// TwinCAT 3 PLC project PLC
// ProgramVersion: 3.1.4023.0
// libraries:
//   Tc2_MC2, * (Beckhoff Automation GmbH)
//   Tc2_MC2_Drive, * (Beckhoff Automation GmbH)
//   Tc2_Standard, * (Beckhoff Automation GmbH)
//   Tc2_System, * (Beckhoff Automation GmbH)
//   Tc2_TcpIp, * (Beckhoff Automation GmbH)
//   Tc2_Utilities, * (Beckhoff Automation GmbH)
//   Tc3_Database, * (Beckhoff Automation GmbH)
//   Tc3_EventLogger, * (Beckhoff Automation GmbH)
//   Tc3_Module, * (Beckhoff Automation GmbH)
// project tree:
//   DUTs/ConveyorSystem/ ST_CPI_Module.TcDUT
//   DUTs/OPC_UA/ OPC_CNC_Data_Collection.TcDUT
//   DUTs/PyADS/ ST_PyADS_Test.TcDUT
//   DUTs/RGB/ ST_RGB_In.TcDUT, ST_RGB_Light.TcDUT, ST_RGB_Out.TcDUT
//   DUTs/ ST_Dut_Data.TcDUT
//   DUTs/Vise/ E_ViseSocketState.TcDUT, E_Vise_State.TcDUT, E_Vise_Command.TcDUT, ST_Order.TcDUT, ST_Vise_Sensors.TcDUT, ST_Vise_Status.TcDUT
//   DUTs/Executer/ E_Executer_State.TcDUT
//   GVLs/ GVL_Ads.TcGVL, GVL_CNC1.TcGVL, GVL_CNC2.TcGVL, GVL_CNC3.TcGVL, GVL_Constant.TcGVL, GVL_ConveyorSystem.TcGVL, GVL_IO.TcGVL, GVL_IO_CNC1.TcGVL, GVL_Main.TcGVL, GVL_Palette.TcGVL, GVL_Python.TcGVL, GVL_RFID.TcGVL, GVL_Safety.TcGVL
//   / PlcTask.TcTTO
//   POUs/ Blink.TcPOU, ConveyorSystem.TcPOU, InitTCPIP.TcPOU, MAIN.TcPOU, SafetyPRG.TcPOU, SQL_Test.TcPOU, Test.TcPOU
//   POUs/CNC_1/ CNC_1.TcPOU
//   POUs/CNC_2/ CNC_2.TcPOU
//   POUs/CNC_3/ CNC_3.TcPOU
//   POUs/FBs/AWEA/DUTs/ ST_AWEA_In.TcDUT, ST_AWEA_Out.TcDUT
//   POUs/FBs/AWEA/ FB_AWEA.TcPOU
//   POUs/FBs/BTL/DUTs/ U_to_dint.TcDUT
//   POUs/FBs/BTL/ FB_BTL1AR0.TcPOU
//   POUs/FBs/Camera/ FB_TCP_IP_Comm.TcPOU
//   POUs/FBs/CNC_Servo/DUTs/ E_CncServoCommand.TcTLEO
//   POUs/FBs/CNC_Servo/ FB_CNC_Servo.TcPOU
//   POUs/FBs/FanucCNC/DUTs/ E_CNC_Robot_Command.TcDUT, E_CNC_Robot_Path.TcTLEO, E_CNC_Robot_Programs.TcTLEO, E_Lifter.TcDUT, ST_CNC_Robot_Control.TcDUT, ST_CNC_Robot_Status.TcDUT, U_CNC_Fanuc_Input.TcDUT, U_CNC_Fanuc_Output.TcDUT
//   POUs/FBs/FanucCNC/ FB_Fanuc_CNC.TcPOU
//   POUs/FBs/FanucKardex/DUTs/ E_Kardex_Robot_Command.TcDUT, E_Kardex_Robot_Programs.TcTLEO, ST_Kardex_Robot_Control.TcDUT, ST_Kardex_Robot_Status.TcDUT, U_Kardex_Fanuc_Input.TcDUT, U_Kardex_Fanuc_Output.TcDUT
//   POUs/FBs/FanucKardex/ FB_Fanuc_Kardex.TcPOU
//   POUs/FBs/Fanuc/DUTs/ E_Robot_Command.TcDUT, E_Robot_Programs.TcTLEO, ST_Robot_Control.TcDUT (not stored), ST_Robot_Status.TcDUT, U_Fanuc_Input.TcDUT, U_Fanuc_Output.TcDUT
//   POUs/FBs/Fanuc/ FB_Fanuc.TcPOU
//   POUs/FBs/ FB_Conveyor.TcPOU, FB_Door.TcPOU, FB_Server.TcPOU, FB_SQL.TcPOU, FB_Vise_Station.TcPOU
//   POUs/FBs/ID200/DUTs/ E_CarrierType.TcTLEO, E_Command.TcTLEO, E_TagStatus.TcTLEO, RawToUlint.TcDUT, ST_Active_RFIDs.TcDUT, ST_Tag_Data.TcDUT, WordToBytes.TcDUT
//   POUs/FBs/ID200/ FB_ID200.TcPOU
//   POUs/FBs/Lift/ FB_Lift.TcPOU
//   POUs/FBs/MPS/DUTs/ U_to_int.TcDUT
//   POUs/FBs/MPS/ FB_MPS100.TcPOU
//   POUs/FBs/MySQL/NextVise/DUTs/ ST_ParaVal_GetNextVise.TcDUT
//   POUs/FBs/MySQL/NextVise/ FB_SP_spGetNextVise.TcPOU
//   POUs/FBs/MySQL/SetViseState/DUTs/ ST_ParaVal_SetViseStae.TcDUT
//   POUs/FBs/MySQL/SetViseState/ FB_SP_spSetViseStae.TcPOU
//   POUs/FBs/MySQL/UpdateVise/DUTs/ ST_ParaVal_UpdateVise.TcDUT
//   POUs/FBs/MySQL/UpdateVise/ FB_SP_spUpdateVise.TcPOU
//   POUs/FBs/Pneumatics/ FB_Bistabil.TcPOU, FB_Stopper.TcPOU, FB_Stopper2.TcPOU
//   POUs/FBs/Router/ FB_Router.TcPOU
//   POUs/FBs/ServoVise/DUTs/ E_ServoVise_Command.TcTLEO, E_ViseJawState.TcTLEO
//   POUs/FBs/ServoVise/ FB_ServoVise.TcPOU, FB_TorqueCheck.TcPOU
//   POUs/FBs/Utilities/ FB_CommandLineExecuter.TcPOU, FB_FullCycleTime.TcPOU, FB_GenPulse.TcPOU, FB_Not_SmartLight.TcPOU, FB_RGB_Light.TcPOU, FB_TcEvent.TcPOU, FB_UpsC69xx.TcPOU, FB_UserLed.TcPOU, FB_WorkLight.TcPOU
//   POUs/Robot7AxisStation/ Robot7AxisProgram.TcPOU
//   POUs/RobotKardexStation/ RobotKardexProgram.TcPOU
//   POUs/RobotViseStation/ RobotCncProgram.TcPOU, ViseProgram.TcPOU
//   POUs/Temp/Fanuc/ E_Fanuc_Program.TcDUT, ST_FanucReq.TcDUT, ST_Fanuc_Alarm_In.TcDUT, ST_Fanuc_Alarm_Out.TcDUT, ST_Fanuc_Area_In.TcDUT, ST_Fanuc_Control_In.TcDUT, ST_Fanuc_Control_Out.TcDUT, ST_Fanuc_Data_In.TcDUT, ST_Fanuc_Data_Out.TcDUT, ST_Fanuc_DIO_In.TcDUT, ST_Fanuc_Emergency_In.TcDUT, ST_Fanuc_HandShake_In.TcDUT, ST_Fanuc_Handshake_Out.TcDUT, ST_Fanuc_In.TcDUT, ST_Fanuc_ManPos.TcDUT, ST_Fanuc_Out.TcDUT, ST_Fanuc_Press_Out.TcDUT, ST_Fanuc_Prog_In.TcDUT, ST_Fanuc_Prog_Out.TcDUT, U_Fanuc_In.TcDUT, U_Fanuc_Out.TcDUT
//   POUs/Temp/ FB_ContiRobot.TcPOU, Robot.TcPOU
//   POUs/UploadingStation/ UploadingProgram.TcPOU
// real-time tasks:
//   TASK PlcTask: cycle T#10ms, priority 20, ADS port 350
//   TASK ProfiNET: cycle T#16ms, priority 25, ADS port 351
//   TASK Job Task: cycle default, priority 32
// motion (NC):
//   TASK NC-Task 1 SAF: cycle T#2ms, priority 4, ADS port 501
//   TASK NC-Task 1 SVB: cycle T#10ms, priority 8, ADS port 511
//   AXIS Axis 1 (id 1)
//     Dynamic: Acceleration=6.6163, Deceleration=6.6163, Jerk=19.8489
//     Velo: RefSearch=0.044108688151042, RefSync=0.044108688151042, SlowManual=0.220543440755208, FastManual=4, Fast=4.41086881510417, Maximum=4.41087
//     OtherSettings: AllowMotionCmdToSlave=true
//     encoder EncType=8
//       EncPara: ScaleFactorNumerator=0.04, ScaleFactorDenominator=1048576, MaxCount=#xffffffff
//         TimeComp: TimeCompMode=1
//     drive DrvType=9
//       DrvPara: MaxCount=#xffffffff, DriveControlDWord=#x00030100
//         Analog: VeloReferenz=4.85195569661458, VeloScale=1.02400649589962, TorqueSetpointScale=10, ScaleFactorActTorque=0.1
//         TimeComp: TaskDelayCycles=1
//     controller CtrType=1
//       CtrPara: PriorControlFactor=1
//         Observer: BandWidth=20
//   AXIS Axis 2 (id 2)
//     Dynamic: Acceleration=6.6163, Deceleration=6.6163, Jerk=19.8489
//     Velo: RefSearch=0.044108688151042, RefSync=0.044108688151042, SlowManual=0.220543440755208, FastManual=4, Fast=4.41086881510417, Maximum=4.41087
//     OtherSettings: AllowMotionCmdToSlave=true
//     encoder EncType=8
//       EncPara: ScaleFactorNumerator=0.04, ScaleFactorDenominator=1048576, MaxCount=#xffffffff
//         TimeComp: TimeCompMode=1
//     drive DrvType=9
//       DrvPara: MaxCount=#xffffffff, DriveControlDWord=#x00030100
//         Analog: VeloReferenz=4.85195569661458, VeloScale=1.02400649589962, TorqueSetpointScale=10, ScaleFactorActTorque=0.1
//         TimeComp: TaskDelayCycles=1
//     controller CtrType=1
//       CtrPara: PriorControlFactor=1
//         Observer: BandWidth=20
//   AXIS Axis 3 (id 3)
//     Dynamic: Acceleration=6.6163, Deceleration=6.6163, Jerk=19.8489
//     Velo: RefSearch=0.044108688151042, RefSync=0.044108688151042, SlowManual=0.220543440755208, FastManual=4, Fast=4.41086881510417, Maximum=4.41087
//     OtherSettings: AllowMotionCmdToSlave=true
//     encoder EncType=8
//       EncPara: ScaleFactorNumerator=0.04, ScaleFactorDenominator=1048576, MaxCount=#xffffffff
//         TimeComp: TimeCompMode=1
//     drive DrvType=9
//       DrvPara: MaxCount=#xffffffff, DriveControlDWord=#x00030100
//         Analog: VeloReferenz=4.85195569661458, VeloScale=1.02400649589962, TorqueSetpointScale=10, ScaleFactorActTorque=0.1
//         TimeComp: TaskDelayCycles=1
//     controller CtrType=1
//       CtrPara: PriorControlFactor=1
//         Observer: BandWidth=20
// I/O:
//   DEVICE Device 1 (RT-Ethernet Adapter)
//   DEVICE Fanuc_Vise, AmsNetId 192.168.81.10.5.1
//     Box 1 (CU2508) [CU2508 Ethernet Port]
//     Box 2 (FANUC R-30iB V8.20) [FANUC R-30iB V8.20]
//   DEVICE Fanuc_7Axis, AmsNetId 192.168.81.10.6.1
//     Box 3 (CU2508) [CU2508 Ethernet Port]
//     Box 4 (FANUC R-30iB V8.20) [FANUC R-30iB V8.20]
//   DEVICE Fanuc_Kardex, AmsNetId 192.168.81.10.7.1
//     Box 5 (CU2508) [CU2508 Ethernet Port]
//     Box 6 (FANUC R-30iB V8.20) [FANUC R-30iB V8.20]
//   DEVICE CNC_1, AmsNetId 192.168.81.10.8.1
//     Box 7 (CU2508) [CU2508 Ethernet Port]
//     Drive 9 (AX5106-0000-0214) [AX5106-0000-0214 EtherCAT Drive (SoE, 1 Ch.)]
//       Term 16 (AX5805) [AX5805 (Safety Drive Option)]
//         modules: Module 1 (Safety Process Data, 1 axis), Module 2 (Standard Process Data, 1 axis)
//       Term 18 (EL9011) [EL9011 End Terminal]
//     Box 10 (BNI ECT-508-105-Z015) [BNI ECT-508-105-Z015 (BNI0077)]
//       modules: Module 1 (IOL_I_4byte), Module 2 (STD_IN_1bit), Module 3 (STD_IN_1bit), Module 4 (STD_IN_1bit), Module 5 (STD_IN_1bit), Module 6 (STD_IN_1bit), Module 7 (STD_IN_1bit), Module 8 (STD_IN_1bit)
//     Term 11 (EK1100) [EK1100 EtherCAT Coupler (2A E-Bus)]
//       Term 12 (EL6910) [EL6910, TwinSAFE PLC]
//       Term 13 (EL1809) [EL1809 16Ch. Dig. Input 24V, 3ms]
//       Term 14 (EL2809-0015) [EL2809-0015 16Ch. Dig. Output 24V DC, 0.35A, not short-circuit proof]
//       Term 11 (EL9011) [EL9011 End Terminal]
//     Box 15 (EP1957-0022) [EP1957, 8Ch. Safety Input 24V, 4Ch. Safety Output 24V, 0.5A, TwinSAFE]
//       modules: Module 1 (FSOE), Module 2 (FSOUT), Module 3 (DEVICEIO), Module 4 (FSLOGIC)
//   DEVICE CNC_2, AmsNetId 192.168.81.10.9.1
//     Box 18 (CU2508) [CU2508 Ethernet Port]
//     Drive 19 (AX5106-0000-0214) [AX5106-0000-0214 EtherCAT Drive (SoE, 1 Ch.)]
//       Term 20 (AX5805) [AX5805 (Safety Drive Option)]
//         modules: Module 1 (Safety Process Data, 1 axis), Module 2 (Standard Process Data, 1 axis)
//       Term 10 (EL9011) [EL9011 End Terminal]
//     Box 21 (BNI ECT-508-105-Z015) [BNI ECT-508-105-Z015 (BNI0077)]
//       modules: Module 1 (IOL_I_4byte), Module 2 (STD_IN_1bit), Module 3 (STD_IN_1bit), Module 4 (STD_IN_1bit), Module 5 (STD_IN_1bit), Module 6 (STD_IN_1bit), Module 7 (STD_IN_1bit), Module 8 (STD_IN_1bit)
//     Term 22 (EK1100) [EK1100 EtherCAT Coupler (2A E-Bus)]
//       Term 23 (EL6910) [EL6910, TwinSAFE PLC]
//       Term 24 (EL1809) [EL1809 16Ch. Dig. Input 24V, 3ms]
//       Term 25 (EL2809) [EL2809 16Ch. Dig. Output 24V, 0.5A]
//       Term 11 (EL9011) [EL9011 End Terminal]
//     Box 26 (EP1957-0022) [EP1957, 8Ch. Safety Input 24V, 4Ch. Safety Output 24V, 0.5A, TwinSAFE]
//       modules: Module 1 (FSOE), Module 2 (FSOUT), Module 3 (DEVICEIO), Module 4 (FSLOGIC)
//   DEVICE CNC_3, AmsNetId 192.168.81.10.10.1
//     Box 29 (CU2508) [CU2508 Ethernet Port]
//     Drive 30 (AX5106-0000-0214) [AX5106-0000-0214 EtherCAT Drive (SoE, 1 Ch.)]
//       Term 31 (AX5805) [AX5805 (Safety Drive Option)]
//         modules: Module 1 (Safety Process Data, 1 axis), Module 2 (Standard Process Data, 1 axis)
//       Term 10 (EL9011) [EL9011 End Terminal]
//     Box 32 (BNI ECT-508-105-Z015) [BNI ECT-508-105-Z015 (BNI0077)]
//       modules: Module 1 (IOL_I_4byte), Module 2 (STD_IN_1bit), Module 3 (STD_IN_1bit), Module 4 (STD_IN_1bit), Module 5 (STD_IN_1bit), Module 6 (STD_IN_1bit), Module 7 (STD_IN_1bit), Module 8 (STD_IN_1bit)
//     Term 33 (EK1100) [EK1100 EtherCAT Coupler (2A E-Bus)]
//       Term 34 (EL6910) [EL6910, TwinSAFE PLC]
//       Term 35 (EL1809) [EL1809 16Ch. Dig. Input 24V, 3ms]
//       Term 36 (EL2809) [EL2809 16Ch. Dig. Output 24V, 0.5A]
//       Term 11 (EL9011) [EL9011 End Terminal]
//     Box 37 (EP1957-0022) [EP1957, 8Ch. Safety Input 24V, 4Ch. Safety Output 24V, 0.5A, TwinSAFE]
//       modules: Module 1 (FSOE), Module 2 (FSOUT), Module 3 (DEVICEIO), Module 4 (FSLOGIC)
//   DEVICE Main, AmsNetId 192.168.81.10.11.1
//     Box 40 (CU2508) [CU2508 Ethernet Port]
//     Term 41 (EK1100) [EK1100 EtherCAT Coupler (2A E-Bus)]
//       Term 42 (EL6910) [EL6910, TwinSAFE PLC]
//       Term 43 (EL1918) [EL1918, 8Ch. Safety Input 24V, TwinSAFE]
//         modules: Module 1 (FSOE), Module 2 (FSLOGIC)
//       Term 44 (EL1904) [EL1904, 4 Ch. Safety Input 24V, TwinSAFE]
//         modules: Module 1 (FSOES)
//       Term 45 (EL1904) [EL1904, 4 Ch. Safety Input 24V, TwinSAFE]
//         modules: Module 1 (FSOES)
//       Term 46 (EL2904) [EL2904, 4 Ch. Safety Output 24V, 0.5A, TwinSAFE]
//         modules: Module 1 (FSOES), Module 2 (DO)
//       Term 47 (EL2904) [EL2904, 4 Ch. Safety Output 24V, 0.5A, TwinSAFE]
//         modules: Module 1 (FSOES), Module 2 (DO)
//       Term 48 (EL1809) [EL1809 16Ch. Dig. Input 24V, 3ms]
//       Term 49 (EL1809) [EL1809 16Ch. Dig. Input 24V, 3ms]
//       Term 50 (EL1809) [EL1809 16Ch. Dig. Input 24V, 3ms]
//       Term 51 (EL2809) [EL2809 16Ch. Dig. Output 24V, 0.5A]
//       Term 52 (EL2809-0015) [EL2809-0015 16Ch. Dig. Output 24V DC, 0.35A, not short-circuit proof]
//       Term 53 (EL9410) [EL9410 E-Bus Power Supplier  (Diagnostics)]
//       Term 54 (EL2809-0015) [EL2809-0015 16Ch. Dig. Output 24V DC, 0.35A, not short-circuit proof]
//       Term 55 (EL6224) [EL6224 (IO Link Master)]
//       Term 56 (EL6224) [EL6224 (IO Link Master)]
//       Term 18 (EL6631) [EL6631 PROFINET IO Controller]
//       Term 36 (EL9011) [EL9011 End Terminal]
//     Term 58 (EK1100) [EK1100 EtherCAT Coupler (2A E-Bus)]
//       Term 59 (EL1918) [EL1918, 8Ch. Safety Input 24V, TwinSAFE]
//         modules: Module 1 (FSOE), Module 2 (FSLOGIC)
//       Term 60 (EL1918) [EL1918, 8Ch. Safety Input 24V, TwinSAFE]
//         modules: Module 1 (FSOE), Module 2 (FSLOGIC)
//       Term 61 (EL1904) [EL1904, 4 Ch. Safety Input 24V, TwinSAFE]
//         modules: Module 1 (FSOES)
//       Term 62 (EL1904) [EL1904, 4 Ch. Safety Input 24V, TwinSAFE]
//         modules: Module 1 (FSOES)
//       Term 63 (EL2904) [EL2904, 4 Ch. Safety Output 24V, 0.5A, TwinSAFE]
//         modules: Module 1 (FSOES), Module 2 (DO)
//       Term 64 (EL2904) [EL2904, 4 Ch. Safety Output 24V, 0.5A, TwinSAFE]
//         modules: Module 1 (FSOES), Module 2 (DO)
//       Term 65 (EL1809) [EL1809 16Ch. Dig. Input 24V, 3ms]
//       Term 66 (EL1809) [EL1809 16Ch. Dig. Input 24V, 3ms]
//       Term 67 (EL1809) [EL1809 16Ch. Dig. Input 24V, 3ms]
//       Term 68 (EL2809-0015) [EL2809-0015 16Ch. Dig. Output 24V DC, 0.35A, not short-circuit proof]
//       Term 69 (EL2809-0015) [EL2809-0015 16Ch. Dig. Output 24V DC, 0.35A, not short-circuit proof]
//       Term 70 (EL9410) [EL9410 E-Bus Power Supplier  (Diagnostics)]
//       Term 71 (EL2809-0015) [EL2809-0015 16Ch. Dig. Output 24V DC, 0.35A, not short-circuit proof]
//       Term 72 (EL2809-0015) [EL2809-0015 16Ch. Dig. Output 24V DC, 0.35A, not short-circuit proof]
//       Term 34 (EL6614) [EL6614 4 Port Switch (Ethernet, CoE)]
//       Term 37 (EL9011) [EL9011 End Terminal]
//     Box 74 (CPX-FB37) [CPX-FB37 Fieldbus module]
//       modules: Module 1 (FB37-RIO), Module 2 (CPI: 16 Byte I/0 Byte O), Module 3 (CPI: 4 Byte I/0 Byte O), Module 4 (MPA1G VMPA1-FB-EMG-8 [8DO]), Module 5 (MPA1G VMPA1-FB-EMG-8 [8DO]), Module 6 (MPA1G VMPA1-FB-EMG-8 [8DO]), Module 7 (MPA1G VMPA1-FB-EMG-8 [8DO]), Module 8 (MPA1G VMPA1-FB-EMG-8 [8DO]), Module 9 (MPA1G VMPA1-FB-EMG-8 [8DO]), Module 10 (MPA1G VMPA1-FB-EMG-8 [8DO]), Module 11 (MPA1G VMPA1-FB-EMG-8 [8DO]), Module 12 (MPA1G VMPA1-FB-EMG-8 [8DO]), Module 13 (MPA1G VMPA1-FB-EMG-8 [8DO]), Module 14 (MPA1G VMPA1-FB-EMG-8 [8DO])
//     Box 75 (BNI ECT-508-105-Z015) [BNI ECT-508-105-Z015 (BNI0077)]
//       modules: Module 1 (IOL_I_2byte), Module 2 (IOL_I_2byte), Module 3 (STD_IN_1bit), Module 4 (STD_IN_1bit), Module 5 (STD_IN_1bit), Module 6 (STD_IN_1bit), Module 7 (STD_IN_1bit), Module 8 (STD_IN_1bit)
//   DEVICE Vise, AmsNetId 192.168.81.10.12.1
//     Term 77 (EK1100) [EK1100 EtherCAT Coupler (2A E-Bus)]
//       Term 78 (EL6070-0033) [EL6070-0033 1Ch. Licence key terminal, individual licences]
//       Term 79 (EL1918) [EL1918, 8Ch. Safety Input 24V, TwinSAFE]
//         modules: Module 2 (FSLOGIC)
//       Term 109 (EL1904) [EL1904, 4 Ch. Safety Input 24V, TwinSAFE]
//         modules: Module 1 (FSOES)
//       Term 110 (EL1904) [EL1904, 4 Ch. Safety Input 24V, TwinSAFE]
//         modules: Module 1 (FSOES)
//       Term 80 (EL2904) [EL2904, 4 Ch. Safety Output 24V, 0.5A, TwinSAFE]
//         modules: Module 1 (FSOES), Module 2 (DO)
//       Term 81 (EL2904) [EL2904, 4 Ch. Safety Output 24V, 0.5A, TwinSAFE]
//         modules: Module 1 (FSOES), Module 2 (DO)
//       Term 82 (EL1809) [EL1809 16Ch. Dig. Input 24V, 3ms]
//       Term 83 (EL1809) [EL1809 16Ch. Dig. Input 24V, 3ms]
//       Term 84 (EL2809) [EL2809 16Ch. Dig. Output 24V, 0.5A]
//       Term 85 (EL6224) [EL6224 (IO Link Master)]
//       Term 86 (EK1110) [EK1110 EtherCAT extension]
//     Box 87 (EasyCAT_RGB_2x8) [EasyCAT_RGB_2x8]
//     Box 88 (CPX-FB37) [CPX-FB37 Fieldbus module]
//       modules: Module 1 (FB37-RIO), Input, Output1, Output2, Output3, Output4, Output5, Output6, Output7
//     Box 89 (CPX-FB37) [CPX-FB37 Fieldbus module]
//       modules: Module 1 (FB37-RIO), Input, Output1, Output2, Output3, Output4, Output5, Output6, Output7
//     Term 90 (EK1100) [EK1100 EtherCAT Coupler (2A E-Bus)]
//       Term 91 (EL1809) [EL1809 16Ch. Dig. Input 24V, 3ms]
//       Term 92 (EL2809-0015) [EL2809-0015 16Ch. Dig. Output 24V DC, 0.35A, not short-circuit proof]
//       Term 19 (EL9011) [EL9011 End Terminal]
//     Box 93 (EP1957-0022) [EP1957, 8Ch. Safety Input 24V, 4Ch. Safety Output 24V, 0.5A, TwinSAFE]
//       modules: Module 1 (FSOE), Module 2 (FSOUT), Module 3 (DEVICEIO), Module 4 (FSLOGIC)
//     Box 94 (EP1957-0022) [EP1957, 8Ch. Safety Input 24V, 4Ch. Safety Output 24V, 0.5A, TwinSAFE]
//       modules: Module 1 (FSOE), Module 2 (FSOUT), Module 3 (DEVICEIO), Module 4 (FSLOGIC)
//   DEVICE Device 2 (EL6631), AmsNetId 192.168.81.10.3.1
//     rfm1 [Bosch Rexroth DAP1,ID 200/C-ETH, no PDEV 3842410060]
//       modules: Term 1 (DAP Module), Data
//     rfm2 [Bosch Rexroth DAP1,ID 200/C-ETH, no PDEV 3842410060]
//       modules: Term 3 (DAP Module), Data
//     rfm3 [Bosch Rexroth DAP1,ID 200/C-ETH, no PDEV 3842410060]
//       modules: Term 5 (DAP Module), Data
//     rfm4 [Bosch Rexroth DAP1,ID 200/C-ETH, no PDEV 3842410060]
//       modules: Term 7 (DAP Module), Data
//     rfm5 [Bosch Rexroth DAP1,ID 200/C-ETH, no PDEV 3842410060]
//       modules: Term 9 (DAP Module), Data
//     rfm6 [Bosch Rexroth DAP1,ID 200/C-ETH, no PDEV 3842410060]
//       modules: Term 11 (DAP Module), Data
//     rfm7 [Bosch Rexroth DAP1,ID 200/C-ETH, no PDEV 3842410060]
//       modules: Term 13 (DAP Module), Data
//     rfm8 [Bosch Rexroth DAP1,ID 200/C-ETH, no PDEV 3842410060]
//       modules: Term 15 (DAP Module), Data
//     rfm9 [Bosch Rexroth DAP1,ID 200/C-ETH, no PDEV 3842410060]
//       modules: Term 17 (DAP Module), Data
//     rfm10 [Bosch Rexroth DAP1,ID 200/C-ETH, no PDEV 3842410060]
//       modules: Term 19 (DAP Module), Data
// variable links:
//   CNC_1 <-> CNC_1/Drive 9 (AX5106-0000-0214)/Term 16 (AX5805)
//     Term 11 (EK1100)/Term 12 (EL6910)/ConnectionOutputs/Message_3 RxPDO <-> Module 1 (Safety Process Data, 1 axis)/Inputs (Statusword)/FSOE
//   CNC_1 <-> CNC_1/Term 11 (EK1100)/Term 12 (EL6910)
//     Box 15 (EP1957-0022)/Module 1 (FSOE)/FSoE Inputs/FSOE <-> ConnectionOutputs/Message_4 RxPDO
//     Box 15 (EP1957-0022)/Module 1 (FSOE)/FSoE Outputs/FSOE <-> ConnectionInputs/Message_4 TxPDO
//     Drive 9 (AX5106-0000-0214)/Term 16 (AX5805)/Module 1 (Safety Process Data, 1 axis)/Outputs (Controlword)/FSOE <-> ConnectionInputs/Message_3 TxPDO
//   CNC_1 <-> Main/Term 41 (EK1100)/Term 42 (EL6910)
//     Term 11 (EK1100)/Term 12 (EL6910)/ConnectionInputs/Message_18 TxPDO <-> ConnectionOutputs/Message_26 RxPDO
//     Term 11 (EK1100)/Term 12 (EL6910)/ConnectionOutputs/Message_18 RxPDO <-> ConnectionInputs/Message_26 TxPDO
//   CNC_2 <-> CNC_2/Box 26 (EP1957-0022)
//     Term 22 (EK1100)/Term 23 (EL6910)/ConnectionOutputs/Message_8 RxPDO <-> Module 1 (FSOE)/FSoE Inputs/FSOE
//   CNC_2 <-> CNC_2/Drive 19 (AX5106-0000-0214)/Term 20 (AX5805)
//     Term 22 (EK1100)/Term 23 (EL6910)/ConnectionInputs/Message_7 TxPDO <-> Module 1 (Safety Process Data, 1 axis)/Outputs (Controlword)/FSOE
//     Term 22 (EK1100)/Term 23 (EL6910)/ConnectionOutputs/Message_7 RxPDO <-> Module 1 (Safety Process Data, 1 axis)/Inputs (Statusword)/FSOE
//   CNC_2 <-> CNC_2/Term 22 (EK1100)/Term 23 (EL6910)
//     Box 26 (EP1957-0022)/Module 1 (FSOE)/FSoE Outputs/FSOE <-> ConnectionInputs/Message_8 TxPDO
//   CNC_2 <-> Main/Term 41 (EK1100)/Term 42 (EL6910)
//     Term 22 (EK1100)/Term 23 (EL6910)/ConnectionOutputs/Message_9 RxPDO <-> ConnectionInputs/Message_28 TxPDO
//   CNC_3 <-> CNC_3/Box 37 (EP1957-0022)
//     Term 33 (EK1100)/Term 34 (EL6910)/ConnectionOutputs/Message_9 RxPDO <-> Module 1 (FSOE)/FSoE Inputs/FSOE
//   CNC_3 <-> CNC_3/Drive 30 (AX5106-0000-0214)/Term 31 (AX5805)
//     Term 33 (EK1100)/Term 34 (EL6910)/ConnectionInputs/Message_8 TxPDO <-> Module 1 (Safety Process Data, 1 axis)/Outputs (Controlword)/FSOE
//     Term 33 (EK1100)/Term 34 (EL6910)/ConnectionOutputs/Message_8 RxPDO <-> Module 1 (Safety Process Data, 1 axis)/Inputs (Statusword)/FSOE
//   CNC_3 <-> CNC_3/Term 33 (EK1100)/Term 34 (EL6910)
//     Box 37 (EP1957-0022)/Module 1 (FSOE)/FSoE Outputs/FSOE <-> ConnectionInputs/Message_9 TxPDO
//   CNC_3 <-> Main/Term 41 (EK1100)/Term 42 (EL6910)
//     Term 33 (EK1100)/Term 34 (EL6910)/ConnectionOutputs/Message_10 RxPDO <-> ConnectionInputs/Message_29 TxPDO
//   Main <-> CNC_2/Term 22 (EK1100)/Term 23 (EL6910)
//     Term 41 (EK1100)/Term 42 (EL6910)/ConnectionOutputs/Message_28 RxPDO <-> ConnectionInputs/Message_9 TxPDO
//   Main <-> CNC_3/Term 33 (EK1100)/Term 34 (EL6910)
//     Term 41 (EK1100)/Term 42 (EL6910)/ConnectionOutputs/Message_29 RxPDO <-> ConnectionInputs/Message_10 TxPDO
//   Main <-> Main/Term 41 (EK1100)/Term 42 (EL6910)
//     Term 41 (EK1100)/Term 43 (EL1918)/Module 1 (FSOE)/FSoE Outputs/FSOE <-> ConnectionInputs/Message_17 TxPDO
//     Term 41 (EK1100)/Term 44 (EL1904)/Module 1 (FSOES)/RxPDO/FSOE <-> ConnectionInputs/Message_3 TxPDO
//     Term 41 (EK1100)/Term 45 (EL1904)/Module 1 (FSOES)/RxPDO/FSOE <-> ConnectionInputs/Message_18 TxPDO
//     Term 41 (EK1100)/Term 46 (EL2904)/Module 1 (FSOES)/RxPDO/FSOE <-> ConnectionInputs/Message_5 TxPDO
//     Term 41 (EK1100)/Term 44 (EL1904)/Module 1 (FSOES)/TxPDO/FSOE <-> ConnectionOutputs/Message_3 RxPDO
//     Term 41 (EK1100)/Term 45 (EL1904)/Module 1 (FSOES)/TxPDO/FSOE <-> ConnectionOutputs/Message_18 RxPDO
//     Term 41 (EK1100)/Term 47 (EL2904)/Module 1 (FSOES)/TxPDO/FSOE <-> ConnectionOutputs/Message_22 RxPDO
//   Main <-> Main/Term 41 (EK1100)/Term 43 (EL1918)
//     Term 41 (EK1100)/Term 42 (EL6910)/ConnectionOutputs/Message_17 RxPDO <-> Module 1 (FSOE)/FSoE Inputs/FSOE
//   Main <-> Main/Term 41 (EK1100)/Term 46 (EL2904)
//     Term 41 (EK1100)/Term 42 (EL6910)/ConnectionOutputs/Message_5 RxPDO <-> Module 1 (FSOES)/TxPDO/FSOE
//   Main <-> Main/Term 41 (EK1100)/Term 47 (EL2904)
//     Term 41 (EK1100)/Term 42 (EL6910)/ConnectionInputs/Message_22 TxPDO <-> Module 1 (FSOES)/RxPDO/FSOE
//   Vise <-> Vise/Term 77 (EK1100)/Term 79 (EL1918)
//     Term 77 (EK1100)/Term 80 (EL2904)/Module 1 (FSOES)/RxPDO/FSOE <-> ConnectionInputs/Message_24 TxPDO
//     Term 77 (EK1100)/Term 81 (EL2904)/Module 1 (FSOES)/TxPDO/FSOE <-> ConnectionOutputs/Message_29 RxPDO
//   Vise <-> Vise/Term 77 (EK1100)/Term 80 (EL2904)
//     Term 77 (EK1100)/Term 79 (EL1918)/ConnectionOutputs/Message_24 RxPDO <-> Module 1 (FSOES)/TxPDO/FSOE
//   Vise <-> Vise/Term 77 (EK1100)/Term 81 (EL2904)
//     Term 77 (EK1100)/Term 79 (EL1918)/ConnectionInputs/Message_29 TxPDO <-> Module 1 (FSOES)/RxPDO/FSOE
//   NC-Task 1 SAF/Axes/Axis 1 <-> CNC_1/Drive 9 (AX5106-0000-0214)
//     Drive/Inputs/In/nDataIn1 <-> AT/Following distance
//     Drive/Inputs/In/nDataIn3[0] <-> AT/Torque/force feedback value
//     Drive/Inputs/In/nDcOutputTime <-> InfoData/DcOutputShift
//     Drive/Inputs/In/nState1 <-> AT/Drive status word @bit 8
//     Drive/Inputs/In/nState2 <-> AT/Drive status word
//     Drive/Inputs/In/nState4 @bit 1 <-> WcState/InputToggle
//     Drive/Inputs/In/nState4 <-> WcState/WcState
//     Drive/Outputs/Out/nCtrl1 <-> MDT/Master control word @bit 8
//     Drive/Outputs/Out/nDataOut1 <-> MDT/Position command value
//     Drive/Outputs/Out/nDataOut2 <-> MDT/Velocity command value
//     Drive/Outputs/Out/nDataOut4[0] <-> MDT/Torque/force command value
//     Drive/Outputs/Out/nDataOut5 <-> MDT/High velocity limit value
//     Drive/Outputs/Out/nDataOut6 <-> MDT/Low velocity limit value
//     Enc/Inputs/In/nDataIn1 <-> AT/Position feedback 1 value (motor feedback)
//     Enc/Inputs/In/nDataIn7 <-> AT/Velocity feedback 1 value
//     Enc/Inputs/In/nDcInputTime <-> InfoData/DcInputShift
//     Enc/Inputs/In/nState4 @bit 1 <-> WcState/InputToggle
//     Enc/Inputs/In/nState4 <-> WcState/WcState
//   NC-Task 1 SAF/Axes/Axis 2 <-> CNC_2/Drive 19 (AX5106-0000-0214)
//     Drive/Inputs/In/nDataIn1 <-> AT/Following distance
//     Drive/Inputs/In/nDataIn3[0] <-> AT/Torque/force feedback value
//     Drive/Inputs/In/nDcOutputTime <-> InfoData/DcOutputShift
//     Drive/Inputs/In/nState1 <-> AT/Drive status word @bit 8
//     Drive/Inputs/In/nState2 <-> AT/Drive status word
//     Drive/Inputs/In/nState4 @bit 1 <-> WcState/InputToggle
//     Drive/Inputs/In/nState4 <-> WcState/WcState
//     Drive/Outputs/Out/nCtrl1 <-> MDT/Master control word @bit 8
//     Drive/Outputs/Out/nDataOut1 <-> MDT/Position command value
//     Drive/Outputs/Out/nDataOut2 <-> MDT/Velocity command value
//     Drive/Outputs/Out/nDataOut4[0] <-> MDT/Torque/force command value
//     Drive/Outputs/Out/nDataOut5 <-> MDT/High velocity limit value
//     Drive/Outputs/Out/nDataOut6 <-> MDT/Low velocity limit value
//     Enc/Inputs/In/nDataIn1 <-> AT/Position feedback 1 value (motor feedback)
//     Enc/Inputs/In/nDataIn7 <-> AT/Velocity feedback 1 value
//     Enc/Inputs/In/nDcInputTime <-> InfoData/DcInputShift
//     Enc/Inputs/In/nState4 @bit 1 <-> WcState/InputToggle
//     Enc/Inputs/In/nState4 <-> WcState/WcState
//   NC-Task 1 SAF/Axes/Axis 3 <-> CNC_3/Drive 30 (AX5106-0000-0214)
//     Drive/Inputs/In/nDataIn1 <-> AT/Following distance
//     Drive/Inputs/In/nDataIn3[0] <-> AT/Torque/force feedback value
//     Drive/Inputs/In/nDcOutputTime <-> InfoData/DcOutputShift
//     Drive/Inputs/In/nState1 <-> AT/Drive status word @bit 8
//     Drive/Inputs/In/nState2 <-> AT/Drive status word
//     Drive/Inputs/In/nState4 @bit 1 <-> WcState/InputToggle
//     Drive/Inputs/In/nState4 <-> WcState/WcState
//     Drive/Outputs/Out/nCtrl1 <-> MDT/Master control word @bit 8
//     Drive/Outputs/Out/nDataOut1 <-> MDT/Position command value
//     Drive/Outputs/Out/nDataOut2 <-> MDT/Velocity command value
//     Drive/Outputs/Out/nDataOut4[0] <-> MDT/Torque/force command value
//     Drive/Outputs/Out/nDataOut5 <-> MDT/High velocity limit value
//     Drive/Outputs/Out/nDataOut6 <-> MDT/Low velocity limit value
//     Enc/Inputs/In/nDataIn1 <-> AT/Position feedback 1 value (motor feedback)
//     Enc/Inputs/In/nDataIn7 <-> AT/Velocity feedback 1 value
//     Enc/Inputs/In/nDcInputTime <-> InfoData/DcInputShift
//     Enc/Inputs/In/nState4 @bit 1 <-> WcState/InputToggle
//     Enc/Inputs/In/nState4 <-> WcState/WcState
//   PLC/PLC Instance <-> CNC_1/Box 10 (BNI ECT-508-105-Z015)
//     PlcTask Inputs/CNC_1.fbCncServoVise.fbVisePos.arrRaw[{0..3}] <-> Module 1 (IOL_I_4byte)/TxPDO/input byte {0..3}  (4 links)
//     PlcTask Inputs/CNC_1.fbCncServoVise.fbVisePos.nState <-> IO-Link DeviceState Inputs/Status of IO-Link Port 1
//   PLC/PLC Instance <-> CNC_1/Term 11 (EK1100)/Term 12 (EL6910)
//     PlcTask Inputs/GVL_Safety.i_bLO1_CNC1 <-> StandardInputs/Standard Out Var 21
//     PlcTask Inputs/GVL_Safety.i_bRobotDoorOpened_CNC1 <-> StandardInputs/Standard Out Var 20
//     PlcTask Outputs/GVL_Safety.q_bSafetyErrorAck_Main <-> StandardOutputs/Standard In Var 1
//     PlcTask Outputs/GVL_Safety.q_bSafetyOverrideCnc1 <-> StandardOutputs/Standard In Var 14
//     PlcTask Outputs/GVL_Safety.q_bSafetyRun <-> StandardOutputs/Standard In Var 2
//   PLC/PLC Instance <-> CNC_1/Term 11 (EK1100)/Term 13 (EL1809)
//     PlcTask Inputs/CNC_1.fbCncServoVise.fbLock.i_bBasePos <-> Channel 5/Input
//     PlcTask Inputs/CNC_1.fbCncServoVise.fbLock.i_bWorkPos <-> Channel 6/Input
//     PlcTask Inputs/CNC_1.fbCncServoVise.fbMoveLower.i_bBasePos <-> Channel 4/Input
//     PlcTask Inputs/CNC_1.fbCncServoVise.fbMoveLower.i_bWorkPos <-> Channel 3/Input
//     PlcTask Inputs/CNC_1.fbCncServoVise.fbMoveUpper.i_bBasePos <-> Channel 2/Input
//     PlcTask Inputs/CNC_1.fbCncServoVise.fbMoveUpper.i_bWorkPos <-> Channel 1/Input
//   PLC/PLC Instance <-> CNC_1/Term 11 (EK1100)/Term 14 (EL2809-0015)
//     PlcTask Outputs/CNC_1.fbCncServoVise.fbLock.q_bWorkPos <-> Channel 5/Output
//     PlcTask Outputs/CNC_1.fbCncServoVise.fbMoveLower.q_bBasePos <-> Channel 4/Output
//     PlcTask Outputs/CNC_1.fbCncServoVise.fbMoveLower.q_bWorkPos <-> Channel 3/Output
//     PlcTask Outputs/CNC_1.fbCncServoVise.fbMoveUpper.q_bBasePos <-> Channel 2/Output
//     PlcTask Outputs/CNC_1.fbCncServoVise.fbMoveUpper.q_bWorkPos <-> Channel 1/Output
//     PlcTask Outputs/CNC_1.fbCncServoVise.q_bToolCheckBlower <-> Channel 6/Output
//   PLC/PLC Instance <-> CNC_2/Box 21 (BNI ECT-508-105-Z015)
//     PlcTask Inputs/CNC_2.fbCncServoVise.fbVisePos.arrRaw[{0..3}] <-> Module 1 (IOL_I_4byte)/TxPDO/input byte {0..3}  (4 links)
//     PlcTask Inputs/CNC_2.fbCncServoVise.fbVisePos.nState <-> IO-Link DeviceState Inputs/Status of IO-Link Port 1
//   PLC/PLC Instance <-> CNC_2/Term 22 (EK1100)/Term 23 (EL6910)
//     PlcTask Inputs/GVL_Safety.i_bLO1_CNC2 <-> StandardInputs/Standard Out Var 5
//     PlcTask Inputs/GVL_Safety.i_bRobotDoorOpened_CNC2 <-> StandardInputs/Standard Out Var 6
//     PlcTask Outputs/GVL_Safety.q_bSafetyErrorAck_Main <-> StandardOutputs/Standard In Var 1
//     PlcTask Outputs/GVL_Safety.q_bSafetyOverrideCnc2 <-> StandardOutputs/Standard In Var 4
//     PlcTask Outputs/GVL_Safety.q_bSafetyRun <-> StandardOutputs/Standard In Var 3
//   PLC/PLC Instance <-> CNC_2/Term 22 (EK1100)/Term 24 (EL1809)
//     PlcTask Inputs/CNC_2.fbCncServoVise.fbLock.i_bBasePos <-> Channel 6/Input
//     PlcTask Inputs/CNC_2.fbCncServoVise.fbLock.i_bWorkPos <-> Channel 5/Input
//     PlcTask Inputs/CNC_2.fbCncServoVise.fbMoveLower.i_bBasePos <-> Channel 3/Input
//     PlcTask Inputs/CNC_2.fbCncServoVise.fbMoveLower.i_bWorkPos <-> Channel 4/Input
//     PlcTask Inputs/CNC_2.fbCncServoVise.fbMoveUpper.i_bBasePos <-> Channel 1/Input
//     PlcTask Inputs/CNC_2.fbCncServoVise.fbMoveUpper.i_bWorkPos <-> Channel 2/Input
//   PLC/PLC Instance <-> CNC_2/Term 22 (EK1100)/Term 25 (EL2809)
//     PlcTask Outputs/CNC_2.fbCncServoVise.fbLock.q_bWorkPos <-> Channel 5/Output
//     PlcTask Outputs/CNC_2.fbCncServoVise.fbMoveLower.q_bBasePos <-> Channel 4/Output
//     PlcTask Outputs/CNC_2.fbCncServoVise.fbMoveLower.q_bWorkPos <-> Channel 3/Output
//     PlcTask Outputs/CNC_2.fbCncServoVise.fbMoveUpper.q_bBasePos <-> Channel 2/Output
//     PlcTask Outputs/CNC_2.fbCncServoVise.fbMoveUpper.q_bWorkPos <-> Channel 1/Output
//     PlcTask Outputs/CNC_2.fbCncServoVise.q_bToolCheckBlower <-> Channel 6/Output
//   PLC/PLC Instance <-> CNC_3/Box 32 (BNI ECT-508-105-Z015)
//     PlcTask Inputs/CNC_3.fbCncServoVise.fbVisePos.arrRaw[{0..3}] <-> Module 1 (IOL_I_4byte)/TxPDO/input byte {0..3}  (4 links)
//     PlcTask Inputs/CNC_3.fbCncServoVise.fbVisePos.nState <-> IO-Link DeviceState Inputs/Status of IO-Link Port 1
//   PLC/PLC Instance <-> CNC_3/Term 33 (EK1100)/Term 34 (EL6910)
//     PlcTask Inputs/GVL_Safety.i_bLO1_CNC3 <-> StandardInputs/Standard Out Var 6
//     PlcTask Inputs/GVL_Safety.i_bRobotDoorOpened_CNC3 <-> StandardInputs/Standard Out Var 7
//     PlcTask Outputs/GVL_Safety.q_bSafetyErrorAck_Main <-> StandardOutputs/Standard In Var 2
//     PlcTask Outputs/GVL_Safety.q_bSafetyOverrideCnc3 <-> StandardOutputs/Standard In Var 4
//     PlcTask Outputs/GVL_Safety.q_bSafetyRun <-> StandardOutputs/Standard In Var 3
//   PLC/PLC Instance <-> CNC_3/Term 33 (EK1100)/Term 35 (EL1809)
//     PlcTask Inputs/CNC_3.fbCncServoVise.fbLock.i_bBasePos <-> Channel 6/Input
//     PlcTask Inputs/CNC_3.fbCncServoVise.fbLock.i_bWorkPos <-> Channel 5/Input
//     PlcTask Inputs/CNC_3.fbCncServoVise.fbMoveLower.i_bBasePos <-> Channel 3/Input
//     PlcTask Inputs/CNC_3.fbCncServoVise.fbMoveLower.i_bWorkPos <-> Channel 4/Input
//     PlcTask Inputs/CNC_3.fbCncServoVise.fbMoveUpper.i_bBasePos <-> Channel 1/Input
//     PlcTask Inputs/CNC_3.fbCncServoVise.fbMoveUpper.i_bWorkPos <-> Channel 2/Input
//   PLC/PLC Instance <-> CNC_3/Term 33 (EK1100)/Term 36 (EL2809)
//     PlcTask Outputs/CNC_3.fbCncServoVise.fbLock.q_bWorkPos <-> Channel 5/Output
//     PlcTask Outputs/CNC_3.fbCncServoVise.fbMoveLower.q_bBasePos <-> Channel 4/Output
//     PlcTask Outputs/CNC_3.fbCncServoVise.fbMoveLower.q_bWorkPos <-> Channel 3/Output
//     PlcTask Outputs/CNC_3.fbCncServoVise.fbMoveUpper.q_bBasePos <-> Channel 2/Output
//     PlcTask Outputs/CNC_3.fbCncServoVise.fbMoveUpper.q_bWorkPos <-> Channel 1/Output
//     PlcTask Outputs/CNC_3.fbCncServoVise.q_bToolCheckBlower <-> Channel 6/Output
//   PLC/PLC Instance <-> Device 2 (EL6631)/rfm1
//     PlcTask Inputs/GVL_RFID.fbRFID_Readers[1].PnIoBoxState <-> Inputs/PnIoBoxState
//     PlcTask Inputs/GVL_RFID.fbRFID_Readers[1].arrDataIn[{0..62 step 2}] <-> API/Data/io/Inputs/Response Data[{0..31}]  (32 links)
//     PlcTask Inputs/GVL_RFID.fbRFID_Readers[1].arrDataIn[{1..63 step 2}] <-> API/Data/io/Inputs/Response Data[{0..31}] @bit 8  (32 links)
//     PlcTask Outputs/GVL_RFID.fbRFID_Readers[1].arrDataOut[{0..62 step 2}] <-> API/Data/io/Outputs/Request Data[{0..31}]  (32 links)
//     PlcTask Outputs/GVL_RFID.fbRFID_Readers[1].arrDataOut[{1..63 step 2}] <-> API/Data/io/Outputs/Request Data[{0..31}] @bit 8  (32 links)
//   PLC/PLC Instance <-> Device 2 (EL6631)/rfm10
//     PlcTask Inputs/GVL_RFID.fbRFID_Readers[10].PnIoBoxState <-> Inputs/PnIoBoxState
//     PlcTask Inputs/GVL_RFID.fbRFID_Readers[10].arrDataIn[{0..62 step 2}] <-> API/Data/io/Inputs/Response Data[{0..31}]  (32 links)
//     PlcTask Inputs/GVL_RFID.fbRFID_Readers[10].arrDataIn[{1..63 step 2}] <-> API/Data/io/Inputs/Response Data[{0..31}] @bit 8  (32 links)
//     PlcTask Outputs/GVL_RFID.fbRFID_Readers[10].arrDataOut[{0..62 step 2}] <-> API/Data/io/Outputs/Request Data[{0..31}]  (32 links)
//     PlcTask Outputs/GVL_RFID.fbRFID_Readers[10].arrDataOut[{1..63 step 2}] <-> API/Data/io/Outputs/Request Data[{0..31}] @bit 8  (32 links)
//   PLC/PLC Instance <-> Device 2 (EL6631)/rfm2
//     PlcTask Inputs/GVL_RFID.fbRFID_Readers[2].PnIoBoxState <-> Inputs/PnIoBoxState
//     PlcTask Inputs/GVL_RFID.fbRFID_Readers[2].arrDataIn[{0..62 step 2}] <-> API/Data/io/Inputs/Response Data[{0..31}]  (32 links)
//     PlcTask Inputs/GVL_RFID.fbRFID_Readers[2].arrDataIn[{1..63 step 2}] <-> API/Data/io/Inputs/Response Data[{0..31}] @bit 8  (32 links)
//     PlcTask Outputs/GVL_RFID.fbRFID_Readers[2].arrDataOut[{0..62 step 2}] <-> API/Data/io/Outputs/Request Data[{0..31}]  (32 links)
//     PlcTask Outputs/GVL_RFID.fbRFID_Readers[2].arrDataOut[{1..63 step 2}] <-> API/Data/io/Outputs/Request Data[{0..31}] @bit 8  (32 links)
//   PLC/PLC Instance <-> Device 2 (EL6631)/rfm3
//     PlcTask Inputs/GVL_RFID.fbRFID_Readers[3].PnIoBoxState <-> Inputs/PnIoBoxState
//     PlcTask Inputs/GVL_RFID.fbRFID_Readers[3].arrDataIn[{0..62 step 2}] <-> API/Data/io/Inputs/Response Data[{0..31}]  (32 links)
//     PlcTask Inputs/GVL_RFID.fbRFID_Readers[3].arrDataIn[{1..63 step 2}] <-> API/Data/io/Inputs/Response Data[{0..31}] @bit 8  (32 links)
//     PlcTask Outputs/GVL_RFID.fbRFID_Readers[3].arrDataOut[{0..62 step 2}] <-> API/Data/io/Outputs/Request Data[{0..31}]  (32 links)
//     PlcTask Outputs/GVL_RFID.fbRFID_Readers[3].arrDataOut[{1..63 step 2}] <-> API/Data/io/Outputs/Request Data[{0..31}] @bit 8  (32 links)
//   PLC/PLC Instance <-> Device 2 (EL6631)/rfm4
//     PlcTask Inputs/GVL_RFID.fbRFID_Readers[4].PnIoBoxState <-> Inputs/PnIoBoxState
//     PlcTask Inputs/GVL_RFID.fbRFID_Readers[4].arrDataIn[{0..62 step 2}] <-> API/Data/io/Inputs/Response Data[{0..31}]  (32 links)
//     PlcTask Inputs/GVL_RFID.fbRFID_Readers[4].arrDataIn[{1..63 step 2}] <-> API/Data/io/Inputs/Response Data[{0..31}] @bit 8  (32 links)
//     PlcTask Outputs/GVL_RFID.fbRFID_Readers[4].arrDataOut[{0..62 step 2}] <-> API/Data/io/Outputs/Request Data[{0..31}]  (32 links)
//     PlcTask Outputs/GVL_RFID.fbRFID_Readers[4].arrDataOut[{1..63 step 2}] <-> API/Data/io/Outputs/Request Data[{0..31}] @bit 8  (32 links)
//   PLC/PLC Instance <-> Device 2 (EL6631)/rfm5
//     PlcTask Inputs/GVL_RFID.fbRFID_Readers[5].PnIoBoxState <-> Inputs/PnIoBoxState
//     PlcTask Inputs/GVL_RFID.fbRFID_Readers[5].arrDataIn[{0..62 step 2}] <-> API/Data/io/Inputs/Response Data[{0..31}]  (32 links)
//     PlcTask Inputs/GVL_RFID.fbRFID_Readers[5].arrDataIn[{1..63 step 2}] <-> API/Data/io/Inputs/Response Data[{0..31}] @bit 8  (32 links)
//     PlcTask Outputs/GVL_RFID.fbRFID_Readers[5].arrDataOut[{0..62 step 2}] <-> API/Data/io/Outputs/Request Data[{0..31}]  (32 links)
//     PlcTask Outputs/GVL_RFID.fbRFID_Readers[5].arrDataOut[{1..63 step 2}] <-> API/Data/io/Outputs/Request Data[{0..31}] @bit 8  (32 links)
//   PLC/PLC Instance <-> Device 2 (EL6631)/rfm6
//     PlcTask Inputs/GVL_RFID.fbRFID_Readers[6].PnIoBoxState <-> Inputs/PnIoBoxState
//     PlcTask Inputs/GVL_RFID.fbRFID_Readers[6].arrDataIn[{0..62 step 2}] <-> API/Data/io/Inputs/Response Data[{0..31}]  (32 links)
//     PlcTask Inputs/GVL_RFID.fbRFID_Readers[6].arrDataIn[{1..63 step 2}] <-> API/Data/io/Inputs/Response Data[{0..31}] @bit 8  (32 links)
//     PlcTask Outputs/GVL_RFID.fbRFID_Readers[6].arrDataOut[{0..62 step 2}] <-> API/Data/io/Outputs/Request Data[{0..31}]  (32 links)
//     PlcTask Outputs/GVL_RFID.fbRFID_Readers[6].arrDataOut[{1..63 step 2}] <-> API/Data/io/Outputs/Request Data[{0..31}] @bit 8  (32 links)
//   PLC/PLC Instance <-> Device 2 (EL6631)/rfm7
//     PlcTask Inputs/GVL_RFID.fbRFID_Readers[7].PnIoBoxState <-> Inputs/PnIoBoxState
//     PlcTask Inputs/GVL_RFID.fbRFID_Readers[7].arrDataIn[{0..62 step 2}] <-> API/Data/io/Inputs/Response Data[{0..31}]  (32 links)
//     PlcTask Inputs/GVL_RFID.fbRFID_Readers[7].arrDataIn[{1..63 step 2}] <-> API/Data/io/Inputs/Response Data[{0..31}] @bit 8  (32 links)
//     PlcTask Outputs/GVL_RFID.fbRFID_Readers[7].arrDataOut[{0..62 step 2}] <-> API/Data/io/Outputs/Request Data[{0..31}]  (32 links)
//     PlcTask Outputs/GVL_RFID.fbRFID_Readers[7].arrDataOut[{1..63 step 2}] <-> API/Data/io/Outputs/Request Data[{0..31}] @bit 8  (32 links)
//   PLC/PLC Instance <-> Device 2 (EL6631)/rfm8
//     PlcTask Inputs/GVL_RFID.fbRFID_Readers[8].PnIoBoxState <-> Inputs/PnIoBoxState
//     PlcTask Inputs/GVL_RFID.fbRFID_Readers[8].arrDataIn[{0..62 step 2}] <-> API/Data/io/Inputs/Response Data[{0..31}]  (32 links)
//     PlcTask Inputs/GVL_RFID.fbRFID_Readers[8].arrDataIn[{1..63 step 2}] <-> API/Data/io/Inputs/Response Data[{0..31}] @bit 8  (32 links)
//     PlcTask Outputs/GVL_RFID.fbRFID_Readers[8].arrDataOut[{0..62 step 2}] <-> API/Data/io/Outputs/Request Data[{0..31}]  (32 links)
//     PlcTask Outputs/GVL_RFID.fbRFID_Readers[8].arrDataOut[{1..63 step 2}] <-> API/Data/io/Outputs/Request Data[{0..31}] @bit 8  (32 links)
//   PLC/PLC Instance <-> Device 2 (EL6631)/rfm9
//     PlcTask Inputs/GVL_RFID.fbRFID_Readers[9].PnIoBoxState <-> Inputs/PnIoBoxState
//     PlcTask Inputs/GVL_RFID.fbRFID_Readers[9].arrDataIn[{0..62 step 2}] <-> API/Data/io/Inputs/Response Data[{0..31}]  (32 links)
//     PlcTask Inputs/GVL_RFID.fbRFID_Readers[9].arrDataIn[{1..63 step 2}] <-> API/Data/io/Inputs/Response Data[{0..31}] @bit 8  (32 links)
//     PlcTask Outputs/GVL_RFID.fbRFID_Readers[9].arrDataOut[{0..62 step 2}] <-> API/Data/io/Outputs/Request Data[{0..31}]  (32 links)
//     PlcTask Outputs/GVL_RFID.fbRFID_Readers[9].arrDataOut[{1..63 step 2}] <-> API/Data/io/Outputs/Request Data[{0..31}] @bit 8  (32 links)
//   PLC/PLC Instance <-> Fanuc_7Axis/Box 4 (FANUC R-30iB V8.20)
//     PlcTask Inputs/Robot7AxisProgram.fbRobot.RobotIn.aStdIn <-> IN512/DO00
//     PlcTask Inputs/Robot7AxisProgram.fbRobot.RobotIn.aStdIn @bit 128 <-> IN512/DO01
//     PlcTask Inputs/Robot7AxisProgram.fbRobot.RobotIn.aStdIn @bit 256 <-> IN512/DO02
//     PlcTask Inputs/Robot7AxisProgram.fbRobot.RobotIn.aStdIn @bit 384 <-> IN512/DO03
//     PlcTask Outputs/Robot7AxisProgram.fbRobot.RobotOut.aStdOut <-> OUT512/DI00
//     PlcTask Outputs/Robot7AxisProgram.fbRobot.RobotOut.aStdOut @bit 128 <-> OUT512/DI01
//     PlcTask Outputs/Robot7AxisProgram.fbRobot.RobotOut.aStdOut @bit 256 <-> OUT512/DI02
//     PlcTask Outputs/Robot7AxisProgram.fbRobot.RobotOut.aStdOut @bit 384 <-> OUT512/DI03
//   PLC/PLC Instance <-> Fanuc_Kardex/Box 6 (FANUC R-30iB V8.20)
//     PlcTask Inputs/RobotKardexProgram.fbRobot.RobotIn.aStdIn <-> IN512/DO00
//     PlcTask Inputs/RobotKardexProgram.fbRobot.RobotIn.aStdIn @bit 128 <-> IN512/DO01
//     PlcTask Inputs/RobotKardexProgram.fbRobot.RobotIn.aStdIn @bit 256 <-> IN512/DO02
//     PlcTask Inputs/RobotKardexProgram.fbRobot.RobotIn.aStdIn @bit 384 <-> IN512/DO03
//     PlcTask Outputs/RobotKardexProgram.fbRobot.RobotOut.aStdOut <-> OUT512/DI00
//     PlcTask Outputs/RobotKardexProgram.fbRobot.RobotOut.aStdOut @bit 128 <-> OUT512/DI01
//     PlcTask Outputs/RobotKardexProgram.fbRobot.RobotOut.aStdOut @bit 256 <-> OUT512/DI02
//     PlcTask Outputs/RobotKardexProgram.fbRobot.RobotOut.aStdOut @bit 384 <-> OUT512/DI03
//   PLC/PLC Instance <-> Fanuc_Vise/Box 2 (FANUC R-30iB V8.20)
//     PlcTask Inputs/RobotCncProgram.fbRobot.RobotIn.aStdIn <-> IN512/DO00
//     PlcTask Inputs/RobotCncProgram.fbRobot.RobotIn.aStdIn @bit 128 <-> IN512/DO01
//     PlcTask Inputs/RobotCncProgram.fbRobot.RobotIn.aStdIn @bit 256 <-> IN512/DO02
//     PlcTask Inputs/RobotCncProgram.fbRobot.RobotIn.aStdIn @bit 384 <-> IN512/DO03
//     PlcTask Outputs/RobotCncProgram.fbRobot.RobotOut.aStdOut <-> OUT512/DI00
//     PlcTask Outputs/RobotCncProgram.fbRobot.RobotOut.aStdOut @bit 128 <-> OUT512/DI01
//     PlcTask Outputs/RobotCncProgram.fbRobot.RobotOut.aStdOut @bit 256 <-> OUT512/DI02
//     PlcTask Outputs/RobotCncProgram.fbRobot.RobotOut.aStdOut @bit 384 <-> OUT512/DI03
//   PLC/PLC Instance <-> Main/Box 74 (CPX-FB37)
//     PlcTask Inputs/GVL_ConveyorSystem.i_stSensorHub_0 <-> Module 2 (CPI: 16 Byte I/0 Byte O)/Inputs/Input 0
//     PlcTask Inputs/GVL_ConveyorSystem.i_stSensorHub_1 <-> Module 2 (CPI: 16 Byte I/0 Byte O)/Inputs/Input 1
//     PlcTask Inputs/GVL_ConveyorSystem.i_stSensorHub_10 <-> Module 2 (CPI: 16 Byte I/0 Byte O)/Inputs/Input 10
//     PlcTask Inputs/GVL_ConveyorSystem.i_stSensorHub_11 <-> Module 2 (CPI: 16 Byte I/0 Byte O)/Inputs/Input 11
//     PlcTask Inputs/GVL_ConveyorSystem.i_stSensorHub_12 <-> Module 2 (CPI: 16 Byte I/0 Byte O)/Inputs/Input 12
//     PlcTask Inputs/GVL_ConveyorSystem.i_stSensorHub_13 <-> Module 2 (CPI: 16 Byte I/0 Byte O)/Inputs/Input 13
//     PlcTask Inputs/GVL_ConveyorSystem.i_stSensorHub_14 <-> Module 2 (CPI: 16 Byte I/0 Byte O)/Inputs/Input 14
//     PlcTask Inputs/GVL_ConveyorSystem.i_stSensorHub_15 <-> Module 2 (CPI: 16 Byte I/0 Byte O)/Inputs/Input 15
//     PlcTask Inputs/GVL_ConveyorSystem.i_stSensorHub_16 <-> Module 3 (CPI: 4 Byte I/0 Byte O)/Inputs/Input 0
//     PlcTask Inputs/GVL_ConveyorSystem.i_stSensorHub_17 <-> Module 3 (CPI: 4 Byte I/0 Byte O)/Inputs/Input 1
//     PlcTask Inputs/GVL_ConveyorSystem.i_stSensorHub_18 <-> Module 3 (CPI: 4 Byte I/0 Byte O)/Inputs/Input 2
//     PlcTask Inputs/GVL_ConveyorSystem.i_stSensorHub_19 <-> Module 3 (CPI: 4 Byte I/0 Byte O)/Inputs/Input 3
//     PlcTask Inputs/GVL_ConveyorSystem.i_stSensorHub_2 <-> Module 2 (CPI: 16 Byte I/0 Byte O)/Inputs/Input 2
//     PlcTask Inputs/GVL_ConveyorSystem.i_stSensorHub_3 <-> Module 2 (CPI: 16 Byte I/0 Byte O)/Inputs/Input 3
//     PlcTask Inputs/GVL_ConveyorSystem.i_stSensorHub_4 <-> Module 2 (CPI: 16 Byte I/0 Byte O)/Inputs/Input 4
//     PlcTask Inputs/GVL_ConveyorSystem.i_stSensorHub_5 <-> Module 2 (CPI: 16 Byte I/0 Byte O)/Inputs/Input 5
//     PlcTask Inputs/GVL_ConveyorSystem.i_stSensorHub_6 <-> Module 2 (CPI: 16 Byte I/0 Byte O)/Inputs/Input 6
//     PlcTask Inputs/GVL_ConveyorSystem.i_stSensorHub_7 <-> Module 2 (CPI: 16 Byte I/0 Byte O)/Inputs/Input 7
//     PlcTask Inputs/GVL_ConveyorSystem.i_stSensorHub_8 <-> Module 2 (CPI: 16 Byte I/0 Byte O)/Inputs/Input 8
//     PlcTask Inputs/GVL_ConveyorSystem.i_stSensorHub_9 <-> Module 2 (CPI: 16 Byte I/0 Byte O)/Inputs/Input 9
//     PlcTask Outputs/GVL_ConveyorSystem.q_bS1 <-> Module 9 (MPA1G VMPA1-FB-EMG-8 [8DO])/Outputs/Output 3
//     PlcTask Outputs/GVL_ConveyorSystem.q_bS10 <-> Module 10 (MPA1G VMPA1-FB-EMG-8 [8DO])/Outputs/Output 2
//     PlcTask Outputs/GVL_ConveyorSystem.q_bS11 <-> Module 10 (MPA1G VMPA1-FB-EMG-8 [8DO])/Outputs/Output 5
//     PlcTask Outputs/GVL_ConveyorSystem.q_bS12 <-> Module 10 (MPA1G VMPA1-FB-EMG-8 [8DO])/Outputs/Output 4
//     PlcTask Outputs/GVL_ConveyorSystem.q_bS13 <-> Module 10 (MPA1G VMPA1-FB-EMG-8 [8DO])/Outputs/Output 7
//     PlcTask Outputs/GVL_ConveyorSystem.q_bS14 <-> Module 10 (MPA1G VMPA1-FB-EMG-8 [8DO])/Outputs/Output 6
//     PlcTask Outputs/GVL_ConveyorSystem.q_bS15 <-> Module 11 (MPA1G VMPA1-FB-EMG-8 [8DO])/Outputs/Output 1
//     PlcTask Outputs/GVL_ConveyorSystem.q_bS16 <-> Module 11 (MPA1G VMPA1-FB-EMG-8 [8DO])/Outputs/Output 0
//     PlcTask Outputs/GVL_ConveyorSystem.q_bS17 <-> Module 11 (MPA1G VMPA1-FB-EMG-8 [8DO])/Outputs/Output 3
//     PlcTask Outputs/GVL_ConveyorSystem.q_bS18 <-> Module 11 (MPA1G VMPA1-FB-EMG-8 [8DO])/Outputs/Output 2
//     PlcTask Outputs/GVL_ConveyorSystem.q_bS19 <-> Module 11 (MPA1G VMPA1-FB-EMG-8 [8DO])/Outputs/Output 5
//     PlcTask Outputs/GVL_ConveyorSystem.q_bS2 <-> Module 9 (MPA1G VMPA1-FB-EMG-8 [8DO])/Outputs/Output 2
//     PlcTask Outputs/GVL_ConveyorSystem.q_bS20 <-> Module 11 (MPA1G VMPA1-FB-EMG-8 [8DO])/Outputs/Output 4
//     PlcTask Outputs/GVL_ConveyorSystem.q_bS21 <-> Module 11 (MPA1G VMPA1-FB-EMG-8 [8DO])/Outputs/Output 7
//     PlcTask Outputs/GVL_ConveyorSystem.q_bS22 <-> Module 11 (MPA1G VMPA1-FB-EMG-8 [8DO])/Outputs/Output 6
//     PlcTask Outputs/GVL_ConveyorSystem.q_bS23 <-> Module 12 (MPA1G VMPA1-FB-EMG-8 [8DO])/Outputs/Output 1
//     PlcTask Outputs/GVL_ConveyorSystem.q_bS24 <-> Module 12 (MPA1G VMPA1-FB-EMG-8 [8DO])/Outputs/Output 0
//     PlcTask Outputs/GVL_ConveyorSystem.q_bS25 <-> Module 12 (MPA1G VMPA1-FB-EMG-8 [8DO])/Outputs/Output 3
//     PlcTask Outputs/GVL_ConveyorSystem.q_bS26 <-> Module 12 (MPA1G VMPA1-FB-EMG-8 [8DO])/Outputs/Output 2
//     PlcTask Outputs/GVL_ConveyorSystem.q_bS27 <-> Module 12 (MPA1G VMPA1-FB-EMG-8 [8DO])/Outputs/Output 5
//     PlcTask Outputs/GVL_ConveyorSystem.q_bS28 <-> Module 12 (MPA1G VMPA1-FB-EMG-8 [8DO])/Outputs/Output 4
//     PlcTask Outputs/GVL_ConveyorSystem.q_bS29 <-> Module 12 (MPA1G VMPA1-FB-EMG-8 [8DO])/Outputs/Output 7
//     PlcTask Outputs/GVL_ConveyorSystem.q_bS3 <-> Module 9 (MPA1G VMPA1-FB-EMG-8 [8DO])/Outputs/Output 5
//     PlcTask Outputs/GVL_ConveyorSystem.q_bS30 <-> Module 12 (MPA1G VMPA1-FB-EMG-8 [8DO])/Outputs/Output 6
//     PlcTask Outputs/GVL_ConveyorSystem.q_bS31 <-> Module 13 (MPA1G VMPA1-FB-EMG-8 [8DO])/Outputs/Output 1
//     PlcTask Outputs/GVL_ConveyorSystem.q_bS32 <-> Module 13 (MPA1G VMPA1-FB-EMG-8 [8DO])/Outputs/Output 0
//     PlcTask Outputs/GVL_ConveyorSystem.q_bS4 <-> Module 9 (MPA1G VMPA1-FB-EMG-8 [8DO])/Outputs/Output 4
//     PlcTask Outputs/GVL_ConveyorSystem.q_bS5 <-> Module 9 (MPA1G VMPA1-FB-EMG-8 [8DO])/Outputs/Output 7
//     PlcTask Outputs/GVL_ConveyorSystem.q_bS6 <-> Module 9 (MPA1G VMPA1-FB-EMG-8 [8DO])/Outputs/Output 6
//     PlcTask Outputs/GVL_ConveyorSystem.q_bS7 <-> Module 10 (MPA1G VMPA1-FB-EMG-8 [8DO])/Outputs/Output 1
//     PlcTask Outputs/GVL_ConveyorSystem.q_bS8 <-> Module 10 (MPA1G VMPA1-FB-EMG-8 [8DO])/Outputs/Output 0
//     PlcTask Outputs/GVL_ConveyorSystem.q_bS9 <-> Module 10 (MPA1G VMPA1-FB-EMG-8 [8DO])/Outputs/Output 3
//     PlcTask Outputs/GVL_ConveyorSystem.q_bZ10_12 <-> Module 6 (MPA1G VMPA1-FB-EMG-8 [8DO])/Outputs/Output 3
//     PlcTask Outputs/GVL_ConveyorSystem.q_bZ10_14 <-> Module 6 (MPA1G VMPA1-FB-EMG-8 [8DO])/Outputs/Output 2
//     PlcTask Outputs/GVL_ConveyorSystem.q_bZ11_12 <-> Module 6 (MPA1G VMPA1-FB-EMG-8 [8DO])/Outputs/Output 5
//     PlcTask Outputs/GVL_ConveyorSystem.q_bZ11_14 <-> Module 6 (MPA1G VMPA1-FB-EMG-8 [8DO])/Outputs/Output 4
//     PlcTask Outputs/GVL_ConveyorSystem.q_bZ12_12 <-> Module 6 (MPA1G VMPA1-FB-EMG-8 [8DO])/Outputs/Output 7
//     PlcTask Outputs/GVL_ConveyorSystem.q_bZ12_14 <-> Module 6 (MPA1G VMPA1-FB-EMG-8 [8DO])/Outputs/Output 6
//     PlcTask Outputs/GVL_ConveyorSystem.q_bZ13_12 <-> Module 7 (MPA1G VMPA1-FB-EMG-8 [8DO])/Outputs/Output 1
//     PlcTask Outputs/GVL_ConveyorSystem.q_bZ13_14 <-> Module 7 (MPA1G VMPA1-FB-EMG-8 [8DO])/Outputs/Output 0
//     PlcTask Outputs/GVL_ConveyorSystem.q_bZ14_12 <-> Module 7 (MPA1G VMPA1-FB-EMG-8 [8DO])/Outputs/Output 3
//     PlcTask Outputs/GVL_ConveyorSystem.q_bZ14_14 <-> Module 7 (MPA1G VMPA1-FB-EMG-8 [8DO])/Outputs/Output 2
//     PlcTask Outputs/GVL_ConveyorSystem.q_bZ15_12 <-> Module 7 (MPA1G VMPA1-FB-EMG-8 [8DO])/Outputs/Output 5
//     PlcTask Outputs/GVL_ConveyorSystem.q_bZ15_14 <-> Module 7 (MPA1G VMPA1-FB-EMG-8 [8DO])/Outputs/Output 4
//     PlcTask Outputs/GVL_ConveyorSystem.q_bZ16_12 <-> Module 7 (MPA1G VMPA1-FB-EMG-8 [8DO])/Outputs/Output 7
//     PlcTask Outputs/GVL_ConveyorSystem.q_bZ16_14 <-> Module 7 (MPA1G VMPA1-FB-EMG-8 [8DO])/Outputs/Output 6
//     PlcTask Outputs/GVL_ConveyorSystem.q_bZ17_12 <-> Module 8 (MPA1G VMPA1-FB-EMG-8 [8DO])/Outputs/Output 1
//     PlcTask Outputs/GVL_ConveyorSystem.q_bZ17_14 <-> Module 8 (MPA1G VMPA1-FB-EMG-8 [8DO])/Outputs/Output 0
//     PlcTask Outputs/GVL_ConveyorSystem.q_bZ18_12 <-> Module 8 (MPA1G VMPA1-FB-EMG-8 [8DO])/Outputs/Output 3
//     PlcTask Outputs/GVL_ConveyorSystem.q_bZ18_14 <-> Module 8 (MPA1G VMPA1-FB-EMG-8 [8DO])/Outputs/Output 2
//     PlcTask Outputs/GVL_ConveyorSystem.q_bZ19_12 <-> Module 8 (MPA1G VMPA1-FB-EMG-8 [8DO])/Outputs/Output 5
//     PlcTask Outputs/GVL_ConveyorSystem.q_bZ19_14 <-> Module 8 (MPA1G VMPA1-FB-EMG-8 [8DO])/Outputs/Output 4
//     PlcTask Outputs/GVL_ConveyorSystem.q_bZ1_12 <-> Module 4 (MPA1G VMPA1-FB-EMG-8 [8DO])/Outputs/Output 1
//     PlcTask Outputs/GVL_ConveyorSystem.q_bZ1_14 <-> Module 4 (MPA1G VMPA1-FB-EMG-8 [8DO])/Outputs/Output 0
//     PlcTask Outputs/GVL_ConveyorSystem.q_bZ20_12 <-> Module 8 (MPA1G VMPA1-FB-EMG-8 [8DO])/Outputs/Output 7
//     PlcTask Outputs/GVL_ConveyorSystem.q_bZ20_14 <-> Module 8 (MPA1G VMPA1-FB-EMG-8 [8DO])/Outputs/Output 6
//     PlcTask Outputs/GVL_ConveyorSystem.q_bZ21_12 <-> Module 9 (MPA1G VMPA1-FB-EMG-8 [8DO])/Outputs/Output 1
//     PlcTask Outputs/GVL_ConveyorSystem.q_bZ21_14 <-> Module 9 (MPA1G VMPA1-FB-EMG-8 [8DO])/Outputs/Output 0
//     PlcTask Outputs/GVL_ConveyorSystem.q_bZ2_12 <-> Module 4 (MPA1G VMPA1-FB-EMG-8 [8DO])/Outputs/Output 3
//     PlcTask Outputs/GVL_ConveyorSystem.q_bZ2_14 <-> Module 4 (MPA1G VMPA1-FB-EMG-8 [8DO])/Outputs/Output 2
//     PlcTask Outputs/GVL_ConveyorSystem.q_bZ3_12 <-> Module 4 (MPA1G VMPA1-FB-EMG-8 [8DO])/Outputs/Output 5
//     PlcTask Outputs/GVL_ConveyorSystem.q_bZ3_14 <-> Module 4 (MPA1G VMPA1-FB-EMG-8 [8DO])/Outputs/Output 4
//     PlcTask Outputs/GVL_ConveyorSystem.q_bZ4_12 <-> Module 4 (MPA1G VMPA1-FB-EMG-8 [8DO])/Outputs/Output 7
//     PlcTask Outputs/GVL_ConveyorSystem.q_bZ4_14 <-> Module 4 (MPA1G VMPA1-FB-EMG-8 [8DO])/Outputs/Output 6
//     PlcTask Outputs/GVL_ConveyorSystem.q_bZ5_12 <-> Module 5 (MPA1G VMPA1-FB-EMG-8 [8DO])/Outputs/Output 1
//     PlcTask Outputs/GVL_ConveyorSystem.q_bZ5_14 <-> Module 5 (MPA1G VMPA1-FB-EMG-8 [8DO])/Outputs/Output 0
//     PlcTask Outputs/GVL_ConveyorSystem.q_bZ6_12 <-> Module 5 (MPA1G VMPA1-FB-EMG-8 [8DO])/Outputs/Output 3
//     PlcTask Outputs/GVL_ConveyorSystem.q_bZ6_14 <-> Module 5 (MPA1G VMPA1-FB-EMG-8 [8DO])/Outputs/Output 2
//     PlcTask Outputs/GVL_ConveyorSystem.q_bZ7_12 <-> Module 5 (MPA1G VMPA1-FB-EMG-8 [8DO])/Outputs/Output 5
//     PlcTask Outputs/GVL_ConveyorSystem.q_bZ7_14 <-> Module 5 (MPA1G VMPA1-FB-EMG-8 [8DO])/Outputs/Output 4
//     PlcTask Outputs/GVL_ConveyorSystem.q_bZ8_12 <-> Module 5 (MPA1G VMPA1-FB-EMG-8 [8DO])/Outputs/Output 7
//     PlcTask Outputs/GVL_ConveyorSystem.q_bZ8_14 <-> Module 5 (MPA1G VMPA1-FB-EMG-8 [8DO])/Outputs/Output 6
//     PlcTask Outputs/GVL_ConveyorSystem.q_bZ9_12 <-> Module 6 (MPA1G VMPA1-FB-EMG-8 [8DO])/Outputs/Output 1
//     PlcTask Outputs/GVL_ConveyorSystem.q_bZ9_14 <-> Module 6 (MPA1G VMPA1-FB-EMG-8 [8DO])/Outputs/Output 0
//   PLC/PLC Instance <-> Main/Box 75 (BNI ECT-508-105-Z015)
//     PlcTask Inputs/GVL_IO.fbGripperPos1.arrRaw[0] <-> Module 1 (IOL_I_2byte)/TxPDO/input byte 0
//     PlcTask Inputs/GVL_IO.fbGripperPos1.arrRaw[1] <-> Module 1 (IOL_I_2byte)/TxPDO/input byte 1
//     PlcTask Inputs/GVL_IO.fbGripperPos2.arrRaw[0] <-> Module 2 (IOL_I_2byte)/TxPDO/input byte 0
//     PlcTask Inputs/GVL_IO.fbGripperPos2.arrRaw[1] <-> Module 2 (IOL_I_2byte)/TxPDO/input byte 1
//     PlcTask Inputs/GVL_IO.fbGripperPos1.nState <-> IO-Link DeviceState Inputs/Status of IO-Link Port 1
//     PlcTask Inputs/GVL_IO.fbGripperPos2.nState <-> IO-Link DeviceState Inputs/Status of IO-Link Port 2
//   PLC/PLC Instance <-> Main/Term 41 (EK1100)/Term 42 (EL6910)
//     PlcTask Inputs/GVL_Safety.i_bLO1EDMErr_Main <-> StandardInputs/Standard Out Var 15
//     PlcTask Inputs/GVL_Safety.i_bLO2EDMErr_Main <-> StandardInputs/Standard Out Var 16
//     PlcTask Inputs/GVL_Safety.i_bLO1_Main <-> StandardInputs/Standard Out Var 13
//     PlcTask Inputs/GVL_Safety.i_bLO2_Main <-> StandardInputs/Standard Out Var 14
//     PlcTask Inputs/GVL_Safety.i_bSafetyGroupComErr_Main <-> StandardInputs/Standard Out Var 10
//     PlcTask Inputs/GVL_Safety.i_bSafetyGroupFBErr_Main <-> StandardInputs/Standard Out Var 11
//     PlcTask Inputs/GVL_Safety.i_bSafetyGroupOtherErr_Main <-> StandardInputs/Standard Out Var 12
//     PlcTask Outputs/GVL_Safety.q_bBlink <-> StandardOutputs/Standard In Var 8
//     PlcTask Outputs/GVL_Safety.q_bCellEmptyAck_Main <-> StandardOutputs/Standard In Var 9
//     PlcTask Outputs/GVL_Safety.q_bSafetyErrorAck_Main <-> StandardOutputs/Standard In Var 1
//     PlcTask Outputs/GVL_Safety.q_bSafetyMasterOn_Main <-> StandardOutputs/Standard In Var 7
//     PlcTask Outputs/GVL_Safety.q_bSafetyRun <-> StandardOutputs/Standard In Var 2
//   PLC/PLC Instance <-> Main/Term 41 (EK1100)/Term 48 (EL1809)
//     PlcTask Inputs/GVL_IO.i_bConveyor_{1..11}_Ok <-> Channel {1..11}/Input  (11 links)
//     PlcTask Inputs/GVL_IO.i_bTerm48_Ch{12..16} <-> Channel {12..16}/Input  (5 links)
//   PLC/PLC Instance <-> Main/Term 41 (EK1100)/Term 49 (EL1809)
//     PlcTask Inputs/GVL_IO.i_bDoorClosed_Kardex <-> Channel 9/Input
//     PlcTask Inputs/GVL_IO.i_bDoorClosed_Main <-> Channel 12/Input
//     PlcTask Inputs/GVL_IO.i_bDoorRequest_Kardex <-> Channel 11/Input
//     PlcTask Inputs/GVL_IO.i_bDoorRequest_Main <-> Channel 14/Input
//     PlcTask Inputs/GVL_IO.i_bEMYStop{10..17} <-> Channel {1..8}/Input  (8 links)
//     PlcTask Inputs/GVL_IO.i_bMasterOn_Kardex <-> Channel 10/Input
//     PlcTask Inputs/GVL_IO.i_bMasterOn_Main <-> Channel 13/Input
//     PlcTask Inputs/GVL_IO.i_bTerm49_Ch15 <-> Channel 15/Input
//     PlcTask Inputs/GVL_IO.i_bTerm49_Ch16 <-> Channel 16/Input
//   PLC/PLC Instance <-> Main/Term 41 (EK1100)/Term 50 (EL1809)
//     PlcTask Inputs/GVL_IO.i_bErrorAckBtn_Main <-> Channel 2/Input
//     PlcTask Inputs/GVL_IO.i_bTest03 <-> Channel 3/Input
//     PlcTask Inputs/GVL_IO.i_bTest_01 <-> Channel 1/Input
//     PlcTask Inputs/GVL_IO.i_bTest_Down <-> Channel 7/Input
//     PlcTask Inputs/GVL_IO.i_bTest_Stop <-> Channel 6/Input
//     PlcTask Inputs/GVL_IO.i_bTest_Up <-> Channel 5/Input
//   PLC/PLC Instance <-> Main/Term 41 (EK1100)/Term 51 (EL2809)
//     PlcTask Outputs/GVL_IO.q_bDoorRequestLED_Kardex <-> Channel 2/Output
//     PlcTask Outputs/GVL_IO.q_bDoorRequestLED_Main <-> Channel 4/Output
//     PlcTask Outputs/GVL_IO.q_bMasterOnLED_Kardex <-> Channel 1/Output
//     PlcTask Outputs/GVL_IO.q_bMasterOnLED_Main <-> Channel 3/Output
//   PLC/PLC Instance <-> Main/Term 41 (EK1100)/Term 54 (EL2809-0015)
//     PlcTask Outputs/GVL_IO.q_bConveyor_{1..11} <-> Channel {1..11}/Output  (11 links)
//   PLC/PLC Instance <-> Main/Term 58 (EK1100)/Term 60 (EL1918)
//     PlcTask Inputs/GVL_IO.i_nBusState <-> InfoData/State
//   PLC/PLC Instance <-> Vise/Box 87 (EasyCAT_RGB_2x8)
//     PlcTask Inputs/GVL_Main.fbRgbLights.i_stRGB_In/LifeSig <-> Inputs/LifeSignal
//     PlcTask Inputs/GVL_Main.fbRgbLights.i_stRGB_In/Resp <-> Inputs/Response
//     PlcTask Outputs/GVL_Main.fbRgbLights.q_stRGB_Out/Command <-> Outputs/Command
//     PlcTask Outputs/GVL_Main.fbRgbLights.q_stRGB_Out/LifeSig <-> Outputs/LifeSignal
//     PlcTask Outputs/GVL_Main.fbRgbLights.q_stRGB_Out/arrRGB[10] <-> Outputs/RGB_10
//     PlcTask Outputs/GVL_Main.fbRgbLights.q_stRGB_Out/arrRGB[11] <-> Outputs/RGB_11
//     PlcTask Outputs/GVL_Main.fbRgbLights.q_stRGB_Out/arrRGB[12] <-> Outputs/RGB_12
//     PlcTask Outputs/GVL_Main.fbRgbLights.q_stRGB_Out/arrRGB[13] <-> Outputs/RGB_13
//     PlcTask Outputs/GVL_Main.fbRgbLights.q_stRGB_Out/arrRGB[14] <-> Outputs/RGB_14
//     PlcTask Outputs/GVL_Main.fbRgbLights.q_stRGB_Out/arrRGB[15] <-> Outputs/RGB_15
//     PlcTask Outputs/GVL_Main.fbRgbLights.q_stRGB_Out/arrRGB[16] <-> Outputs/RGB_16
//     PlcTask Outputs/GVL_Main.fbRgbLights.q_stRGB_Out/arrRGB[17] <-> Outputs/RGB_17
//     PlcTask Outputs/GVL_Main.fbRgbLights.q_stRGB_Out/arrRGB[18] <-> Outputs/RGB_18
//     PlcTask Outputs/GVL_Main.fbRgbLights.q_stRGB_Out/arrRGB[19] <-> Outputs/RGB_19
//     PlcTask Outputs/GVL_Main.fbRgbLights.q_stRGB_Out/arrRGB[1] <-> Outputs/RGB_01
//     PlcTask Outputs/GVL_Main.fbRgbLights.q_stRGB_Out/arrRGB[20] <-> Outputs/RGB_20
//     PlcTask Outputs/GVL_Main.fbRgbLights.q_stRGB_Out/arrRGB[21] <-> Outputs/RGB_21
//     PlcTask Outputs/GVL_Main.fbRgbLights.q_stRGB_Out/arrRGB[22] <-> Outputs/RGB_22
//     PlcTask Outputs/GVL_Main.fbRgbLights.q_stRGB_Out/arrRGB[23] <-> Outputs/RGB_23
//     PlcTask Outputs/GVL_Main.fbRgbLights.q_stRGB_Out/arrRGB[24] <-> Outputs/RGB_24
//     PlcTask Outputs/GVL_Main.fbRgbLights.q_stRGB_Out/arrRGB[2] <-> Outputs/RGB_02
//     PlcTask Outputs/GVL_Main.fbRgbLights.q_stRGB_Out/arrRGB[3] <-> Outputs/RGB_03
//     PlcTask Outputs/GVL_Main.fbRgbLights.q_stRGB_Out/arrRGB[4] <-> Outputs/RGB_04
//     PlcTask Outputs/GVL_Main.fbRgbLights.q_stRGB_Out/arrRGB[5] <-> Outputs/RGB_05
//     PlcTask Outputs/GVL_Main.fbRgbLights.q_stRGB_Out/arrRGB[6] <-> Outputs/RGB_06
//     PlcTask Outputs/GVL_Main.fbRgbLights.q_stRGB_Out/arrRGB[7] <-> Outputs/RGB_07
//     PlcTask Outputs/GVL_Main.fbRgbLights.q_stRGB_Out/arrRGB[8] <-> Outputs/RGB_08
//     PlcTask Outputs/GVL_Main.fbRgbLights.q_stRGB_Out/arrRGB[9] <-> Outputs/RGB_09
//   PLC/PLC Instance <-> Vise/Box 88 (CPX-FB37)
//     PlcTask Inputs/GVL_IO.i_stViseStationSensors_{1..7} <-> Input/Inputs/Input {0..12 step 2}  (7 links)
//     PlcTask Inputs/GVL_IO.i_stViseStationSensors_{1..7} @bit 8 <-> Input/Inputs/Input {1..13 step 2}  (7 links)
//     PlcTask Outputs/GVL_Main.fbViseStation[1].fbStopper_In.q_bWorkPos <-> Output3/Outputs/Output 0
//     PlcTask Outputs/GVL_Main.fbViseStation[2].fbStopper_In.q_bWorkPos <-> Output3/Outputs/Output 4
//     PlcTask Outputs/GVL_Main.fbViseStation[3].fbStopper_In.q_bWorkPos <-> Output4/Outputs/Output 0
//     PlcTask Outputs/GVL_Main.fbViseStation[4].fbStopper_In.q_bWorkPos <-> Output4/Outputs/Output 4
//     PlcTask Outputs/GVL_Main.fbViseStation[5].fbStopper_In.q_bWorkPos <-> Output5/Outputs/Output 0
//     PlcTask Outputs/GVL_Main.fbViseStation[6].fbStopper_In.q_bWorkPos <-> Output5/Outputs/Output 4
//     PlcTask Outputs/GVL_Main.fbViseStation[7].fbStopper_In.q_bWorkPos <-> Output6/Outputs/Output 0
//     PlcTask Outputs/GVL_Main.fbViseStation[1].fbStopper_Out.q_bWorkPos <-> Output3/Outputs/Output 2
//     PlcTask Outputs/GVL_Main.fbViseStation[2].fbStopper_Out.q_bWorkPos <-> Output3/Outputs/Output 6
//     PlcTask Outputs/GVL_Main.fbViseStation[3].fbStopper_Out.q_bWorkPos <-> Output4/Outputs/Output 2
//     PlcTask Outputs/GVL_Main.fbViseStation[4].fbStopper_Out.q_bWorkPos <-> Output4/Outputs/Output 6
//     PlcTask Outputs/GVL_Main.fbViseStation[5].fbStopper_Out.q_bWorkPos <-> Output5/Outputs/Output 2
//     PlcTask Outputs/GVL_Main.fbViseStation[6].fbStopper_Out.q_bWorkPos <-> Output5/Outputs/Output 6
//     PlcTask Outputs/GVL_Main.fbViseStation[7].fbStopper_Out.q_bWorkPos <-> Output6/Outputs/Output 2
//     PlcTask Outputs/GVL_Main.fbViseStation[1].fbVise.q_bBasePos <-> Output1/Outputs/Output 1
//     PlcTask Outputs/GVL_Main.fbViseStation[2].fbVise.q_bBasePos <-> Output1/Outputs/Output 3
//     PlcTask Outputs/GVL_Main.fbViseStation[3].fbVise.q_bBasePos <-> Output1/Outputs/Output 5
//     PlcTask Outputs/GVL_Main.fbViseStation[4].fbVise.q_bBasePos <-> Output1/Outputs/Output 7
//     PlcTask Outputs/GVL_Main.fbViseStation[5].fbVise.q_bBasePos <-> Output2/Outputs/Output 1
//     PlcTask Outputs/GVL_Main.fbViseStation[6].fbVise.q_bBasePos <-> Output2/Outputs/Output 3
//     PlcTask Outputs/GVL_Main.fbViseStation[7].fbVise.q_bBasePos <-> Output2/Outputs/Output 5
//     PlcTask Outputs/GVL_Main.fbViseStation[1].fbVise.q_bWorkPos <-> Output1/Outputs/Output 0
//     PlcTask Outputs/GVL_Main.fbViseStation[2].fbVise.q_bWorkPos <-> Output1/Outputs/Output 2
//     PlcTask Outputs/GVL_Main.fbViseStation[3].fbVise.q_bWorkPos <-> Output1/Outputs/Output 4
//     PlcTask Outputs/GVL_Main.fbViseStation[4].fbVise.q_bWorkPos <-> Output1/Outputs/Output 6
//     PlcTask Outputs/GVL_Main.fbViseStation[5].fbVise.q_bWorkPos <-> Output2/Outputs/Output 0
//     PlcTask Outputs/GVL_Main.fbViseStation[6].fbVise.q_bWorkPos <-> Output2/Outputs/Output 2
//     PlcTask Outputs/GVL_Main.fbViseStation[7].fbVise.q_bWorkPos <-> Output2/Outputs/Output 4
//   PLC/PLC Instance <-> Vise/Box 89 (CPX-FB37)
//     PlcTask Inputs/GVL_IO.i_stViseStationSensors_{8..14} <-> Input/Inputs/Input {0..12 step 2}  (7 links)
//     PlcTask Inputs/GVL_IO.i_stViseStationSensors_{8..14} @bit 8 <-> Input/Inputs/Input {1..13 step 2}  (7 links)
//     PlcTask Outputs/GVL_Main.fbViseStation[10].fbStopper_In.q_bWorkPos <-> Output4/Outputs/Output 0
//     PlcTask Outputs/GVL_Main.fbViseStation[11].fbStopper_In.q_bWorkPos <-> Output4/Outputs/Output 4
//     PlcTask Outputs/GVL_Main.fbViseStation[12].fbStopper_In.q_bWorkPos <-> Output5/Outputs/Output 0
//     PlcTask Outputs/GVL_Main.fbViseStation[13].fbStopper_In.q_bWorkPos <-> Output5/Outputs/Output 4
//     PlcTask Outputs/GVL_Main.fbViseStation[14].fbStopper_In.q_bWorkPos <-> Output6/Outputs/Output 0
//     PlcTask Outputs/GVL_Main.fbViseStation[8].fbStopper_In.q_bWorkPos <-> Output3/Outputs/Output 0
//     PlcTask Outputs/GVL_Main.fbViseStation[9].fbStopper_In.q_bWorkPos <-> Output3/Outputs/Output 4
//     PlcTask Outputs/GVL_Main.fbViseStation[10].fbStopper_Out.q_bWorkPos <-> Output4/Outputs/Output 2
//     PlcTask Outputs/GVL_Main.fbViseStation[11].fbStopper_Out.q_bWorkPos <-> Output4/Outputs/Output 6
//     PlcTask Outputs/GVL_Main.fbViseStation[12].fbStopper_Out.q_bWorkPos <-> Output5/Outputs/Output 2
//     PlcTask Outputs/GVL_Main.fbViseStation[13].fbStopper_Out.q_bWorkPos <-> Output5/Outputs/Output 6
//     PlcTask Outputs/GVL_Main.fbViseStation[14].fbStopper_Out.q_bWorkPos <-> Output6/Outputs/Output 2
//     PlcTask Outputs/GVL_Main.fbViseStation[8].fbStopper_Out.q_bWorkPos <-> Output3/Outputs/Output 2
//     PlcTask Outputs/GVL_Main.fbViseStation[9].fbStopper_Out.q_bWorkPos <-> Output3/Outputs/Output 6
//     PlcTask Outputs/GVL_Main.fbViseStation[10].fbVise.q_bBasePos <-> Output1/Outputs/Output 5
//     PlcTask Outputs/GVL_Main.fbViseStation[11].fbVise.q_bBasePos <-> Output1/Outputs/Output 7
//     PlcTask Outputs/GVL_Main.fbViseStation[12].fbVise.q_bBasePos <-> Output2/Outputs/Output 1
//     PlcTask Outputs/GVL_Main.fbViseStation[13].fbVise.q_bBasePos <-> Output2/Outputs/Output 3
//     PlcTask Outputs/GVL_Main.fbViseStation[14].fbVise.q_bBasePos <-> Output2/Outputs/Output 5
//     PlcTask Outputs/GVL_Main.fbViseStation[8].fbVise.q_bBasePos <-> Output1/Outputs/Output 1
//     PlcTask Outputs/GVL_Main.fbViseStation[9].fbVise.q_bBasePos <-> Output1/Outputs/Output 3
//     PlcTask Outputs/GVL_Main.fbViseStation[10].fbVise.q_bWorkPos <-> Output1/Outputs/Output 4
//     PlcTask Outputs/GVL_Main.fbViseStation[11].fbVise.q_bWorkPos <-> Output1/Outputs/Output 6
//     PlcTask Outputs/GVL_Main.fbViseStation[12].fbVise.q_bWorkPos <-> Output2/Outputs/Output 0
//     PlcTask Outputs/GVL_Main.fbViseStation[13].fbVise.q_bWorkPos <-> Output2/Outputs/Output 2
//     PlcTask Outputs/GVL_Main.fbViseStation[14].fbVise.q_bWorkPos <-> Output2/Outputs/Output 4
//     PlcTask Outputs/GVL_Main.fbViseStation[8].fbVise.q_bWorkPos <-> Output1/Outputs/Output 0
//     PlcTask Outputs/GVL_Main.fbViseStation[9].fbVise.q_bWorkPos <-> Output1/Outputs/Output 2
//   PLC/PLC Instance <-> Vise/Term 77 (EK1100)/Term 79 (EL1918)
//     PlcTask Inputs/GVL_Safety.i_bLO1EDMErr_CNC45 <-> StandardInputs/Standard Out Var 5
//     PlcTask Inputs/GVL_Safety.i_bLO2EDMErr_CNC45 <-> StandardInputs/Standard Out Var 6
//     PlcTask Inputs/GVL_Safety.i_bLO1_CNC45 <-> StandardInputs/Standard Out Var 13
//     PlcTask Inputs/GVL_Safety.i_bLO2_CNC45 <-> StandardInputs/Standard Out Var 14
//     PlcTask Inputs/GVL_Safety.i_bSafetyGroupComErr_CNC45 <-> StandardInputs/Standard Out Var 15
//     PlcTask Inputs/GVL_Safety.i_bSafetyGroupFBErr_CNC45 <-> StandardInputs/Standard Out Var 16
//     PlcTask Inputs/GVL_Safety.i_bSafetyGroupOtherErr_CNC45 <-> StandardInputs/Standard Out Var 17
//     PlcTask Inputs/GVL_Safety.i_bWaitClose_CNC45 <-> StandardInputs/Standard Out Var 28
//     PlcTask Outputs/GVL_Safety.q_bBlink <-> StandardOutputs/Standard In Var 30
//     PlcTask Outputs/GVL_Safety.q_bCellEmptyAck_CNC45 <-> StandardOutputs/Standard In Var 27
//     PlcTask Outputs/GVL_Safety.q_bSafetyErrorAck_CNC45 <-> StandardOutputs/Standard In Var 1
//     PlcTask Outputs/GVL_Safety.q_bSafetyMasterOn_CNC45 <-> StandardOutputs/Standard In Var 3
//     PlcTask Outputs/GVL_Safety.q_bSafetyRun <-> StandardOutputs/Standard In Var 2
//   PLC/PLC Instance <-> Vise/Term 77 (EK1100)/Term 82 (EL1809)
//     PlcTask Inputs/GVL_IO.i_bAirPressureOk <-> Channel 9/Input
//     PlcTask Inputs/GVL_IO.i_bCaptron <-> Channel 11/Input
//     PlcTask Inputs/GVL_IO.i_bCellAck <-> Channel 10/Input
//     PlcTask Inputs/GVL_IO.i_bVisePos1CleanBtn <-> Channel 3/Input
//     PlcTask Inputs/GVL_IO.i_bVisePos2CleanBtn <-> Channel 7/Input
//     PlcTask Inputs/GVL_IO.i_bVisePos1ErrorAckBtn <-> Channel 4/Input
//     PlcTask Inputs/GVL_IO.i_bVisePos2ErrorAckBtn <-> Channel 8/Input
//     PlcTask Inputs/GVL_IO.i_bVisePos1InBtn <-> Channel 1/Input
//     PlcTask Inputs/GVL_IO.i_bVisePos2InBtn <-> Channel 5/Input
//     PlcTask Inputs/GVL_IO.i_bVisePos1RequestBtn <-> Channel 2/Input
//     PlcTask Inputs/GVL_IO.i_bVisePos2RequestBtn <-> Channel 6/Input
//   PLC/PLC Instance <-> Vise/Term 77 (EK1100)/Term 83 (EL1809)
//     PlcTask Inputs/GVL_IO.i_bDoorClosed <-> Channel 9/Input
//     PlcTask Inputs/GVL_IO.i_bDoorRequest <-> Channel 11/Input
//     PlcTask Inputs/GVL_IO.i_bEMYStop{1..6} <-> Channel {1..6}/Input  (6 links)
//     PlcTask Inputs/GVL_IO.i_bMasterOn_CNC45 <-> Channel 10/Input
//   PLC/PLC Instance <-> Vise/Term 77 (EK1100)/Term 84 (EL2809)
//     PlcTask Outputs/GVL_IO.q_bCaptronLED <-> Channel 13/Output
//     PlcTask Outputs/GVL_IO.q_bCellAckLED <-> Channel 12/Output
//     PlcTask Outputs/GVL_IO.q_bDoorLock <-> Channel 11/Output
//     PlcTask Outputs/GVL_IO.q_bDoorRequestLED <-> Channel 2/Output
//     PlcTask Outputs/GVL_IO.q_bMasterOnLED <-> Channel 1/Output
//     PlcTask Outputs/GVL_IO.q_bVise1CleanLED <-> Channel 5/Output
//     PlcTask Outputs/GVL_IO.q_bVise2CleanLED <-> Channel 9/Output
//     PlcTask Outputs/GVL_IO.q_bVise1ErrorAckLED <-> Channel 6/Output
//     PlcTask Outputs/GVL_IO.q_bVise1InLED <-> Channel 3/Output
//     PlcTask Outputs/GVL_IO.q_bVise2InLED <-> Channel 7/Output
//     PlcTask Outputs/GVL_IO.q_bVise1ReqestLED <-> Channel 4/Output
//     PlcTask Outputs/GVL_IO.q_bVise2ErrorAckBtnLED <-> Channel 10/Output
//     PlcTask Outputs/GVL_IO.q_bVise2RequestLED <-> Channel 8/Output
//   PLC/PLC Instance <-> Vise/Term 77 (EK1100)/Term 85 (EL6224)
//     PlcTask Outputs/GVL_Main.fbNotSmartLight.q_bBuzzer <-> IO-Link Port1/Segment 4 -off/on/flash
//     PlcTask Outputs/GVL_Main.fbNotSmartLight.q_bGreenColor <-> IO-Link Port1/Segment 1 -off/on/flash
//     PlcTask Outputs/GVL_Main.fbNotSmartLight.q_bRedColor <-> IO-Link Port1/Segment 3 -off/on/flash
//     PlcTask Outputs/GVL_Main.fbNotSmartLight.q_bYellowColor <-> IO-Link Port1/Segment 2 -off/on/flash
//   PLC/PLC Instance <-> Vise/Term 90 (EK1100)/Term 91 (EL1809)
//     PlcTask Inputs/GVL_IO.i_bCNC4_Door_Closed <-> Channel 2/Input
//     PlcTask Inputs/GVL_IO.i_bCNC4_Door_HW_opened <-> Channel 11/Input
//     PlcTask Inputs/GVL_IO.i_bCNC4_Door_Opened <-> Channel 1/Input
//     PlcTask Inputs/GVL_IO.i_bCNC4_Error <-> Channel 6/Input
//     PlcTask Inputs/GVL_IO.i_bCNC4_M401_Req <-> Channel 8/Input
//     PlcTask Inputs/GVL_IO.i_bCNC4_M402_Req <-> Channel 9/Input
//     PlcTask Inputs/GVL_IO.i_bCNC4_M403_Req <-> Channel 10/Input
//     PlcTask Inputs/GVL_IO.i_bCNC4_Program_End <-> Channel 5/Input
//     PlcTask Inputs/GVL_IO.i_bCNC4_Program_Ready <-> Channel 3/Input
//     PlcTask Inputs/GVL_IO.i_bCNC4_Program_Run <-> Channel 4/Input
//     PlcTask Inputs/GVL_IO.i_bCNC4_Robot_Mode <-> Channel 7/Input
//   PLC/PLC Instance <-> Vise/Term 90 (EK1100)/Term 92 (EL2809-0015)
//     PlcTask Outputs/GVL_IO.q_bCNC4_CleanTool <-> Channel 9/Output
//     PlcTask Outputs/GVL_IO.q_bCNC4_Door_Close <-> Channel 2/Output
//     PlcTask Outputs/GVL_IO.q_bCNC4_Door_Open <-> Channel 1/Output
//     PlcTask Outputs/GVL_IO.q_bCNC4_Fix_Vise <-> Channel 7/Output
//     PlcTask Outputs/GVL_IO.q_bCNC4_M401_Ack <-> Channel 4/Output
//     PlcTask Outputs/GVL_IO.q_bCNC4_M402_Ack <-> Channel 5/Output
//     PlcTask Outputs/GVL_IO.q_bCNC4_M403_Ack <-> Channel 6/Output
//     PlcTask Outputs/GVL_IO.q_bCNC4_Program_Start <-> Channel 3/Output
//     PlcTask Outputs/GVL_IO.q_bCNC4_Release_Vise <-> Channel 8/Output
//   PLC/PLC Instance <-> NC-Task 1 SAF/Axes/Axis 1
//     PlcTask Inputs/CNC_1.fbCncServoVise.fbServoVise.Axis.NcToPlc <-> Outputs/ToPlc
//     PlcTask Outputs/CNC_1.fbCncServoVise.fbServoVise.Axis.PlcToNc <-> Inputs/FromPlc
//   PLC/PLC Instance <-> NC-Task 1 SAF/Axes/Axis 2
//     PlcTask Inputs/CNC_2.fbCncServoVise.fbServoVise.Axis.NcToPlc <-> Outputs/ToPlc
//     PlcTask Outputs/CNC_2.fbCncServoVise.fbServoVise.Axis.PlcToNc <-> Inputs/FromPlc
//   PLC/PLC Instance <-> NC-Task 1 SAF/Axes/Axis 3
//     PlcTask Inputs/CNC_3.fbCncServoVise.fbServoVise.Axis.NcToPlc <-> Outputs/ToPlc
//     PlcTask Outputs/CNC_3.fbCncServoVise.fbServoVise.Axis.PlcToNc <-> Inputs/FromPlc

CONFIGURATION PLC
    RESOURCE PLC ON TwinCAT3
        TASK PlcTask(INTERVAL := T#10ms, PRIORITY := 20);
        PROGRAM MAIN WITH PlcTask : MAIN;
    END_RESOURCE
END_CONFIGURATION

// ---- DUTs/ConveyorSystem/ST_CPI_Module.TcDUT
TYPE ST_CPI_Module :
STRUCT
	Channel_0	:BIT;
	Channel_1	:BIT;
	Channel_2	:BIT;
	Channel_3	:BIT;
	Channel_4	:BIT;
	Channel_5	:BIT;
	Channel_6	:BIT;
	Channel_7	:BIT;
	Channel_8	:BIT;
	Channel_9	:BIT;
	Channel_10	:BIT;
	Channel_11	:BIT;
	Channel_12	:BIT;
	Channel_13	:BIT;
	Channel_14	:BIT;
	Channel_15	:BIT;
END_STRUCT
END_TYPE

// ---- DUTs/OPC_UA/OPC_CNC_Data_Collection.TcDUT
TYPE OPC_CNC_Data_Collection :
	STRUCT
	HeartBeat						:	DINT;		//Heart beat signal with the C# data-exchanger program
	ErrorMessage					:	STRING;		//Error message from the CNC
	ToolTablePath					:	STRING(80);	//Ensure that the "ToolTablePath" variable here is not empty. This path is used for both for the Read and Load triggers
	MagazineTablePath				:	STRING(80); //Ensure that the "MagazineTablePath" variable here is not empty. This path is used for both for the Read and Load triggers
	ProgramPath						:	STRING(80);	//The path to the program to be executed. It may be a direct path to the CNC file? 
	ProgramLoadTrigger				:	BOOL;		//Not yet useable at 2023.11.07.
	ToolTableLoadTrigger			:	BOOL;		//Change the data of the ToolTable file with the name of the path's filename to the name data of the file under the path  "ToolTablePath"
	MagazineTableLoadTrigger		:	BOOL;		//Change the data of the MagazineTable file with the name of the path's filename to the name data of the file under the path  "MagazineTablePath"
	ReadActualToolTable				:	BOOL;		//Reads the actual tool table's content on the CNC and save it to the given path in ToolTablePath
	ReadActualMagazineTable			:	BOOL;		//Reads the actual magazine table's content on the CNC and save it to the given path in MagazineTablePath
	ReadActualTableDone				:	BOOL;	(*	Only true, if the readed data is saved to the target path, AND if the saved data equals to the data to be saved.
													So this way, the saved data is checked
													This bool is both for Tool and Magazine table. *)
	MidwareRequestedShutdown		:	BOOL;	
	ApproveShutdownRequest			:	BOOL;
		{region Machine}
			{region Channels}
				{region 0}
					CutterLocation					: 	ARRAY[0..4] OF LREAL;	//Actual position of the CNC's Axises
					FeedOverride					: 	UDINT;
					//ChannelID						: 	UDINT;
					OperatingMode					: 	STRING;											//Manual, MDI, RFP, SingleStepp, Automatic, Other, Handweel
					{region Program(OBJECT)}
						ProgramCurrentCall			: 	STRING;
						//ExecutionStack				: 	OpcUa_ProgramPositionArrayType;
						{region ExecutionState(OBJECT)}
							CurentState_Program		: 	STRING;//OpcUa_LocalizedText;					//Idle, Running, Stopped, Finished, Error, Interrupted
							//LastTransition_Program		:	OpcUa_LocalizedText;
							StartCNCProgram				:	BOOL;
							StopCNCProgram				:	BOOL;
							CancelCNCProgram			:	BOOL;
							SelectCNCProgramByNodeID	:	BOOL;
							SelectCNCPrograBlockNumber	:	BOOL;
						{endregion}
						ProgramName					: 	STRING;
					{endregion}					 
					RapidOverride					: 	UDINT;
					RapidTraverseActive				: 	BOOL;
					SpeedOverride					: 	UDINT;
				{endregion}
			{endregion}
			{region Control Info}
				;	 
			{endregion}
			{region Error}
				{region AllActiveErrors(OBJECT)}
					{region Channel0ActiveErros(OBJECT)}
						;
					{endregion}
				{endregion}
			{endregion}
			//HostComputerMode	:	BOOL;
			{region ManufacturerExtensions (OBJECT)}
				{region Control Status (OBJECT)}
					ControlStatus_ControlReady				:	BOOL;
					ControlStatus_Error						:	BOOL;
					ControlStatus_PocketAtLoadingPosition	:	INT;
					ControlStatus_RobotModeActive			:	BOOL;
					ControlStatus_T0Active					:	BOOL;
				{endregion}
				{region Door Control}
					DoorControl_CloseDoor			:	BOOL;
					DoorControl_DoorClosed			:	BOOL;
					DoorControl_DoorOpened			:	BOOL;
					DoorControl_OpenDoor			:	BOOL;
					DoorControl_DoorClosing			:	BOOL;
					DoorControl_DoorOpening			:	BOOL;
					DoorControl_Error				:	BOOL;
				{endregion}
				{region Magazine Table}
					MagazineTable_Error				:	BOOL;
					MagazineTable_Ok				:	BOOL;
					MagazineTable_Busy				:	BOOL;
					MagazineTable_Trigger			:	BOOL;
				{endregion}
				{region Miscellaneous functions}
					M401_Acknowledge				:	BOOL;
					M401_Active						:	BOOL;
					M402_Acknowledge				:	BOOL;
					M402_Active						:	BOOL;
					M403_Acknowledge				:	BOOL;
					M403_Active						:	BOOL;
				{endregion}
				{region Tool Table}
					ToolTable_Error					:	BOOL;
					ToolTable_Ok					:	BOOL;
					ToolTable_Busy					:	BOOL;
					ToolTable_Trigger				:	BOOL;
				{endregion}	 
			{endregion}
			{region Manufacturer Info}
				 ;
			{endregion}
			{region Operating Times}
				//ControlUpTime						:	LREAL;
				//MachineUpTime						:	LREAL;
				//ProgramExecutionTime				:	LREAL;
			{endregion}
			{region OperatorInfo}
				;	 
			{endregion}
			{region State}	//Object -  ns-1	i-51001  
				CurrentState_State					: 	STRING;					// NCIsNotConnected, NCIsConnected, NCIsBooted, NCIsInitializing, NCIsAvailable, NCIsShuttingDown
				//LastTransition_State				:	OpcUa_LocalizedText;
			{endregion}
		{endregion}
		{region Server}
			{region Server Status}
				ServerState							:	STRING;	 				// Running, Failed	,NoConfiguration, Suspended, Shutdown, Test, CommunicationFault, Unknown 
			{endregion}
		{endregion}
	END_STRUCT
END_TYPE

// ---- DUTs/PyADS/ST_PyADS_Test.TcDUT
{attribute 'pack_mode' := '1'}
TYPE ST_PyADS_Test :
STRUCT
  	rVar : LREAL;
    rVar2 : REAL;
    iVar : INT;
    iVar2 : ARRAY [1..3] OF DINT;
    sVar : STRING;
END_STRUCT
END_TYPE

// ---- DUTs/RGB/ST_RGB_In.TcDUT
TYPE ST_RGB_In :
STRUCT
	LifeSig				AT %I*			:UINT;
	Resp				AT %i*			:UINT;
END_STRUCT
END_TYPE

// ---- DUTs/RGB/ST_RGB_Light.TcDUT
TYPE ST_RGB_Light :
STRUCT
	nColor1				:UDINT;
	nColor1State		:BOOL;
	nColor2				:UDINT;
	nColor2State		:BOOL;
	nColor3				:UDINT;
	nColor3State		:BOOL;
END_STRUCT
END_TYPE

// ---- DUTs/RGB/ST_RGB_Out.TcDUT
TYPE ST_RGB_Out :
STRUCT
	arrRGB				AT %Q*			:ARRAY[1..24] OF UDINT;
	LifeSig				AT %Q*			:UINT;
	Command				AT %Q*			:UINT;
END_STRUCT
END_TYPE

// ---- DUTs/ST_Dut_Data.TcDUT
TYPE ST_Dut_Data :
STRUCT
	nDutId			: ULINT;			// HERP adatbázis azonosító
	sSerNr			: STRING;			// HERP sorozatszám
	nPaletteId		: INT;				// Paletta sorszám
	nCamFileId		: ULINT;			// HERP CAM fájl azonosító
	nDimX			: REAL;				// Termék X mérete
	nDimY			: REAL;				// Termék Y mérete
	nDimZ			: REAL;				// Termék Z mérete
	nPosX			: REAL;				// Termék X pozíciója a satuba
	nPosY			: REAL;				// Termék Y pozíciója a satuba
	nTorque			: REAL;				// Satu meghúzási nyomaték
	nWeight			: UINT;				// A termék tömege
	bPass			: BOOL;				// Termék minősítés
	bDutInVise		: BOOL;				// Termék a satuban
	bDone			: BOOL;				// EZ van darabérzékelő helyett a CNC-be
	nState			: UINT;				// Termék státusz
	nTarget			: UINT;				// Célállomás
END_STRUCT
END_TYPE
(*
nState:
00.bit		Konvejorra felpakolva
01.bit		Kiemelve CNC-re vár
02.bit		A terék úton a CNC-be
03.bit		CNC forgácsolás kész
04.bit
05.bit
......
14.bit
15.bit
*)

(*
nTarget:
0:	Kardex
1:	CNC 1 Puffer
2:	CNC 1
3:	CNC 2 Puffer
4:	CNC 2
5:	CNC 3 Puffer
6:	CNC 3
7:	Kihordás
*)

// ---- DUTs/Vise/E_ViseSocketState.TcDUT
{attribute 'qualified_only'}
{attribute 'strict'}
TYPE E_ViseSocketState :
(
	ViseInSocket := 0,
	SocketEmpty	:= 1
);
END_TYPE

// ---- DUTs/Vise/E_Vise_State.TcDUT
{attribute 'qualified_only'}
{attribute 'strict'}
TYPE E_Vise_State :
(
	Empty := 0,
	OutForLoad := 1,
	ReadyToCnc := 2,
	InRobotArmBeforeCnc := 3,
	InCnc := 4,
	CncDone := 5,
	InRobotArmAfterCnc := 6,
	WaitingForUnLoad := 7,
	OutForUnload := 8,
	RequestCleaning := 9,
	OutOfService := 10
);
END_TYPE

// ---- DUTs/Vise/E_Vise_Command.TcDUT
{attribute 'qualified_only'}
{attribute 'strict'}
TYPE E_Vise_Command :
(
	Load,
	InProcess,
	UnLoad
);
END_TYPE

// ---- DUTs/Vise/ST_Order.TcDUT
TYPE ST_Order :
STRUCT
	nViseIndex		:BYTE;	// 1-14
	nCncIndex		:BYTE;	// 4,5
END_STRUCT
END_TYPE

// ---- DUTs/Vise/ST_Vise_Sensors.TcDUT
TYPE ST_Vise_Sensors :
STRUCT
	// Robot
	bViseIn					:BIT;	
	bViseOut				:BIT;	
	// Stopper 1
	bStopper_In_Hold		:BIT;
	bStopper_In_Release		:BIT;
	// Stopper 2
	bStopper_Out_Hold		:BIT;
	bStopper_Out_Release	:BIT;
	bInPos					:BIT;
	bOutPos					:BIT;
	
	bViseIsOut				:BIT;
	{attribute 'hide'} 
	_reserved_1			:BIT;
	{attribute 'hide'}
	_reserved_2			:BIT;
	{attribute 'hide'} 
	_reserved_3			:BIT;
	{attribute 'hide'}
	_reserved_4			:BIT;
	{attribute 'hide'} 
	_reserved_5			:BIT;
	{attribute 'hide'}
	_reserved_6			:BIT;
	{attribute 'hide'}
	_reserved_7			:BIT;
END_STRUCT
END_TYPE

// ---- DUTs/Vise/ST_Vise_Status.TcDUT
TYPE ST_Vise_Status :
STRUCT
	eState			:E_Vise_State;		//
	eSocketState	:E_ViseSocketState;
	nInCNC			:BYTE;
	bPass			:BOOL;
	bFail			:BOOL;
	nViseIndex		:USINT; // 1-14
END_STRUCT
END_TYPE

// ---- DUTs/Executer/E_Executer_State.TcDUT
{attribute 'qualified_only'}
{attribute 'strict'}
TYPE E_Executer_State :
(
	Busy := 0,
	Done := 10,
	Error := 20
);
END_TYPE

// ---- POUs/FBs/AWEA/DUTs/ST_AWEA_In.TcDUT
TYPE ST_AWEA_In :
STRUCT
	DoorOpened			:BIT;
	DoorClosed			:BIT;
	ProgReady			:BIT;
	ProgRun				:BIT;
	ProgEnd				:BIT;
	NotError			:BIT;
	Mode				:BIT;
	M401				:BIT;
	M402				:BIT;
	M403				:BIT;
END_STRUCT
END_TYPE

// ---- POUs/FBs/AWEA/DUTs/ST_AWEA_Out.TcDUT
TYPE ST_AWEA_Out :
STRUCT
	DoorOpen			:BIT;
	DoorClose			:BIT;
	Start				:BIT;
	M401_Ack			:BIT;
	M402_Ack			:BIT;
	M403_Ack			:BIT;
END_STRUCT
END_TYPE

// ---- POUs/FBs/BTL/DUTs/U_to_dint.TcDUT
TYPE U_to_dint :
UNION
	arrRaw			: ARRAY [0..3] OF BITARR8;
	nData			: DINT;
END_UNION
END_TYPE

// ---- POUs/FBs/CNC_Servo/DUTs/E_CncServoCommand.TcTLEO
{attribute 'qualified_only'}
{attribute 'strict'}
TYPE E_CncServoCommand :
(
	NoCommand,
	Base,
	MovePos,
	Fixed,
	Release
);
END_TYPE

// ---- POUs/FBs/FanucCNC/DUTs/E_CNC_Robot_Command.TcDUT
{attribute 'qualified_only'}
{attribute 'strict'}
TYPE E_CNC_Robot_Command :
(
	NoCommand 						:= 0,
	Home							:= 1,
	QuickHome						:= 2,
	Wait							:= 3,
	Service							:= 4,
	Pick_Up_CNC 					:= 5,
	Put_Down_CNC					:= 6,
	Pick_Up_Lifter	 				:= 7,
	Put_Down_Lifter 				:= 8,
	Camera_Lifter					:= 9,
	Pick_Up_Master 					:= 10,
	Put_Down_Master					:= 11,
	Pick_Up_Master_From_Lifter		:= 12,
	Put_Down_Master_To_Lifter		:= 13
);
END_TYPE

// ---- POUs/FBs/FanucCNC/DUTs/E_CNC_Robot_Path.TcTLEO
{attribute 'qualified_only'}
{attribute 'strict'}
TYPE E_CNC_Robot_Path :
(
	NoPath,
	Lift1A_to_CNC1,
	Lift1B_to_CNC1,
	CNC1_to_Lift1A,
	CNC1_to_Lift1B,
	Lift2A_to_CNC2,
	Lift2B_to_CNC2,
	CNC2_to_Lift2A,
	CNC2_to_Lift2B,
	Lift3A_to_CNC3,
	Lift3B_to_CNC3,
	CNC3_to_Lift3A,
	CNC3_to_Lift3B
);
END_TYPE

// ---- POUs/FBs/FanucCNC/DUTs/E_CNC_Robot_Programs.TcTLEO
{attribute 'strict'}
{attribute 'to_string'}
TYPE E_CNC_Robot_Programs :
(
	NoCommand					:= 0, 	// Amíg "0"-ás a programszám addig nincs mozgási program végrehajtás, vár…
	Home						:= 1,	// Robot Zóna-6-ba megy és bemozog alaphelyzetbe
	Park						:= 2,	// Robot Zóna-6-ba megy és bemozog parkoló pozícióba.
	Service						:= 3,	// Robot elmegy szerviz pozícióba.
	QuickHome					:= 4,	// Robot aktuális pozícióból elmegy gyors alaphelyzetbe. (A güdelen az aktuális ponton marad a robot.)
	CNC_1_PutDown				:= 11,	// CNC 1-be rakás
	CNC_1_PickUp 				:= 12,	// CNC 1-ből kivétel
	CNC_2_PutDown 				:= 21,	// CNC 2-be rakás
	CNC_2_PickUp 				:= 22,	// CNC 2-ből kivétel
	CNC_3_PutDown 				:= 31,	// CNC 3-ba rakás
	CNC_3_PickUp  				:= 32,	// CNC 3-ból kivétel
	Lifter_1A_PickUp			:= 41,	// Kiemelő 1A-ból kiszedés
	Lifter_1A_PutDown 			:= 42,	// Kiemelő 1A-ba berakás
	Lifter_1B_PickUp			:= 43,	// Kiemelő 1B-ből kiszedés
	Lifter_1B_PutDown 			:= 44,	// Kiemelő 1B-be berakás
	Lifter_2A_PickUp			:= 51,	// Kiemelő 2A-ból kiszedés
	Lifter_2A_PutDown			:= 52,	// Kiemelő 2A-ba berakás
	Lifter_2B_PickUp			:= 53,	// Kiemelő 2B-ből kiszedés
	Lifter_2B_PutDown  			:= 54,	// Kiemelő 2B-be berakás
	Lifter_3A_PickUp			:= 61,	// Kiemelő 3A-ból kiszedés
	Lifter_3A_PutDown  			:= 62,	// Kiemelő 3A-ba berakás
	Lifter_3B_PickUp 			:= 63,	// Kiemelő 3B-ből kiszedés
	Lifter_3B_PutDown 			:= 64,	// Kiemelő 3B-be berakás
	Lifter_1A_Camera			:= 71,	// Kiemelő 1A-nál kamerázás
	Lifter_1B_Camera 			:= 72,	// Kiemelő 1B-nél kamerázás
	Lifter_2A_Camera			:= 73,	// Kiemelő 2A-nál kamerázás
	Lifter_2B_Camera			:= 74,	// Kiemelő 2B-nél kamerázás
	Lifter_3A_Camera			:= 75,	// Kiemelő 3A-nál kamerázás
	Lifter_3B_Camera 			:= 76,	// Kiemelő 3B-nél kamerázás
	Master_Part_PickUp			:= 101,
	Master_Part_PutDown			:= 102,
	Lifter_1A_Master_PickUp		:= 111,
	Lifter_1A_Master_PutDown	:= 112,
	Lifter_1B_Master_PickUp		:= 113,
	Lifter_1B_Master_PutDown	:= 114,
	Lifter_2A_Master_PickUp 	:= 121,
	Lifter_2A_Master_PutDown	:= 122,
	Lifter_2B_Master_PickUp 	:= 123,
	Lifter_2B_Master_PutDown	:= 124,
	Lifter_3A_Master_PickUp		:= 131,
	Lifter_3A_Master_PutDown	:= 132,
	Lifter_3B_Master_PickUp		:= 133,
	Lifter_3B_Master_PutDown 	:= 134
);
END_TYPE

// ---- POUs/FBs/FanucCNC/DUTs/E_Lifter.TcDUT
{attribute 'qualified_only'}
{attribute 'strict'}
TYPE E_Lifter :
(
	Lifter_1A := 0,
	Lifter_1B := 1,
	Lifter_2A := 2,
	Lifter_2B := 3,
	Lifter_3A := 4,
	Lifter_3B := 5
);
END_TYPE

// ---- POUs/FBs/FanucCNC/DUTs/ST_CNC_Robot_Control.TcDUT
TYPE ST_CNC_Robot_Control :
STRUCT
(*-----=== Byte 01 ===-----*)
	bImmediateStop			:BIT;				// 01.1	Immediate stop
	bHold					:BIT;				// 01.2	Temporary stop
	bSafeSpeed				:BIT;				// 01.3	Safe speed
	bCycleStop				:BIT;				// 01.4	Cycle stop
	bReset					:BIT;				// 01.5	External reset
	bStart					:BIT;				// 01.6	Start
	bHome					:BIT;				// 01.7	Return to home position
	bEnable					:BIT;				// 01.8	Operation enable

(*-----=== Byte 02 ===-----*)
//	nProgNumberSelection	:BYTE;
	bPNS1					:BIT;				// 02.1	Program  number selection
	bPNS2					:BIT;				// 02.2	Program  number selection
	bPNS3					:BIT;				// 02.3	Program  number selection
	bPNS4					:BIT;				// 02.4	Program  number selection
	bPNS5					:BIT;				// 02.5	Program  number selection
	bPNS6					:BIT;				// 02.6	Program  number selection
	bPNS7					:BIT;				// 02.7	Program  number selection
	bPNS8					:BIT;				// 02.8	Program  number selection

(*-----=== Byte 03 ===-----*)
	bPnsStrobe				:BIT;				// 03.1	PNS strobe
	bProdStart				:BIT;				// 03.2	Start of automatic operation
	bZoneEnable				:BIT;				// 03.3	Ez mindig jön kivéve ha vész van
	bServiceEnd				:BIT;				// 03.4	Szervíz üzemmód vége
	{attribute 'hide'}
	_reserved_03_05			:BIT;
	{attribute 'hide'}
	_reserved_03_06			:BIT;
	{attribute 'hide'}
	_reserved_03_07			:BIT;		
	{attribute 'hide'}
	_reserved_03_08			:BIT;		
	
(*-----=== Byte 04 ===-----*)
	{attribute 'hide'}
	_reserved_04			:BYTE;				

(*-----=== Byte 05 ===-----*)
	bCNC_1_Reset			:BIT;				// 05.1	Robot CNC-1-be mehet RESET
	bCNC_1_ViseClose_Reset	:BIT;				// 05.2	Robot CNC-1 satu zárva RESET
	bCNC_1_ViseOpen_Reset	:BIT;				// 05.3	Robot CNC-1 satu nyitva RESET
	bCNC_2_Reset			:BIT;				// 05.4	Robot CNC-2-be mehet RESET
	bCNC_2_ViseClose_Reset	:BIT;				// 05.5	Robot CNC-2 satu zárva RESET
	bCNC_2_ViseOpen_Reset	:BIT;				// 05.6	Robot CNC-2 satu nyitva RESET
	bCNC_3_Reset			:BIT;				// 05.7	Robot CNC-3-be mehet RESET
	bCNC_3_ViseClose_Reset	:BIT;				// 05.8	Robot CNC-3 satu zárva RESET
	
(*-----=== Byte 06 ===-----*)
	bCNC_3_ViseOpen_Reset	:BIT;				// 06.1	Robot CNC-3 satu nyitva RESET
	bPalette_1_Reset		:BIT;				// 06.2	Robot Kiemelő 1-hez mehet RESET
	bPalette_2_Reset		:BIT;				// 06.3	Robot Kiemelő 2-höz mehet RESET
	bPalette_3_Reset		:BIT;				// 06.4	Robot Kiemelő 3-hoz mehet RESET
	bGripperClosed_Reset	:BIT;				// 06.5	Robot megfogó zárás RESET
	{attribute 'hide'}
	_reserved_06_06			:BIT;		
	{attribute 'hide'}
	_reserved_06_07			:BIT;	
	{attribute 'hide'}
	_reserved_06_08			:BIT;			
	
(*-----=== Byte 07 ===-----*)
	bNotCorrectPrg_Reset	:BIT;				// 07.1	Nem megfelelő mozgási program RESET
	bNotProductOnRobot_Reset:BIT;				// 07.2	Mozgási program nem hajtható végre, mert a robotnál nincs termék RESET
	bProductOnRobot_Reset	:BIT;				// 07.3	Mozgási program nem hajtható végre, mert a robotnál termék van RESET
	bGripperOpenError_Reset	:BIT;				// 07.4	Megfogó nyitási hiba RESET
	bGripperCloseError_Reset:BIT;				// 07.5	Megfogó zárási hiba RESET
	bOffsetError_Reset		:BIT;				// 07.6 Offset érték hiba RESET
	bWeightError_Reset		:BIT;				// 07.7 Súly érték hiba  RESET
	{attribute 'hide'}
	_reserved_07_08			:BIT;

(*-----=== Byte 08-12 ===-----*)
	{attribute 'hide'}
	_reserved_08_12			:ARRAY [8..12] OF BYTE;

(*-----=== Byte 13 ===-----*)
	bPlcOverride			:BYTE;				// 13. PLC által vezérelt sebesség, 10-100 %
	
(*-----=== Byte 14 ===-----*)
	nProgramNumber			:BYTE;				// 14. Mozgatási műveletek kiválasztása.
	
(*-----=== Byte 15 ===-----*)
	nMode					:BYTE;				// 15. PLC által meghatározott robot üzemmód, 1-2

(*-----=== Byte 16 ===-----*)
	{attribute 'hide'}
	_reserved_16			:BYTE;	
	
(*-----=== Byte 17-18 ===-----*)
	nWeight					:UINT;				// 16. PLC által megadott súly

(*-----=== Byte 19-20 ===-----*)
	{attribute 'hide'}
	_reserved_19_20			:ARRAY [19..20] OF BYTE;	
	
(*-----=== Byte 21-22 ===-----*)
	nOffset_ID				:UINT;				// 21-22. PLC által megadott offszet érték.
	
(*-----=== Byte 23-24 ===-----*)
	nOffset_X_Whole			:INT;				// 23-24. PLC által átadott X tengelyű egész szám offszet érték.
	
(*-----=== Byte 25-26 ===-----*)
	nOffset_X_Fractional	:UINT;				// 25-26. PLC által átadott X tengelyű egész tört offszet érték
	
(*-----=== Byte 27-28 ===-----*)
	nOffset_Y_Whole			:INT;				// 27-28. PLC által átadott Y tengelyű egész szám offszet érték.
	
(*-----=== Byte 29-30 ===-----*)
	nOffset_Y_Fractional	:UINT;				// 29-30. PLC által átadott Y tengelyű egész tört offszet érték	
	
(*-----=== Byte 31-32 ===-----*)
	nOffset_Z_Whole			:INT;				// 31-32. PLC által átadott Z tengelyű egész szám offszet érték.
	
(*-----=== Byte 33-34 ===-----*)
	nOffset_Z_Fractional	:UINT;				// 33-34. PLC által átadott Z tengelyű egész tört offszet érték	
	
(*-----=== Byte 35-36 ===-----*)
	nOffset_W_Whole			:INT;				// 35-36. PLC által átadott W tengelyű egész szám offszet érték.
	
(*-----=== Byte 37-38 ===-----*)
	nOffset_W_Fractional	:UINT;				// 37-38. PLC által átadott W tengelyű egész tört offszet érték
	
(*-----=== Byte 39-40 ===-----*)
	nOffset_P_Whole			:INT;				// 39-40. PLC által átadott P tengelyű egész szám offszet érték.
	
(*-----=== Byte 41-42 ===-----*)
	nOffset_P_Fractional	:UINT;				// 41-42. PLC által átadott P tengelyű egész tört offszet érték	
	
(*-----=== Byte 43-44 ===-----*)
	nOffset_R_Whole			:INT;				// 43-44. PLC által átadott R tengelyű egész szám offszet érték.
	
(*-----=== Byte 45-46 ===-----*)
	nOffset_R_Fractional	:UINT;				// 45-46. PLC által átadott R tengelyű egész tört offszet érték	
	
(*-----=== Byte 47-64 ===-----*)
	{attribute 'hide'}
	_reserved_47_64			:ARRAY [47..64] OF BYTE;				
END_STRUCT
END_TYPE

// ---- POUs/FBs/FanucCNC/DUTs/ST_CNC_Robot_Status.TcDUT
TYPE ST_CNC_Robot_Status :
STRUCT
(*-----=== Byte 01 ===-----*)
	bCommandEnable			:BIT;				// 01.1	During automatic operation
	bSystemReady			:BIT;				// 01.2	Preparation completed
	bProgRun				:BIT;				// 01.3	Program running
	bPaused					:BIT;				// 01.4	Program being interrupted
	bHeld					:BIT;				// 01.5	During temporary stop
	bFault					:BIT;				// 01.6	Alarm
	bHomePos				:BIT;				// 01.7	Home position
	bPendant				:BIT;				// 01.8	Teach pendant enabled

(*-----=== Byte 02 ===-----*)
	bBatteryVoltageDrop		:BIT;				// 02.1	Battery voltage drop
	bBusy					:BIT;				// 02.1	During operation
	bAckSNO1				:BIT;				// 02.1	Selected program number
	bAckSNO2				:BIT;				// 02.2	Selected program number
	bAckSNO3				:BIT;				// 02.3	Selected program number
	bAckSNO4				:BIT;				// 02.4	Selected program number
	bAckSNO5				:BIT;				// 02.5	Selected program number
	bAckSNO6				:BIT;				// 02.6	Selected program number

(*-----=== Byte 03 ===-----*)
	bAckSNO7				:BIT;				// 03.1	Selected program number
	bAckSNO8				:BIT;				// 03.2	Selected program number
	bSnAck					:BIT;				// 03.3	Response signal to PNS
	{attribute 'hide'}
	_reserved_03_04			:BIT;
	bProgramEnd				:BIT;				// 03.5	Robot aktuális programot befejezte
	bProgramRun				:BIT;				// 03.6	Robot aktuális program futásban.
	bAlarm					:BIT;				// 03.7	Robot kűldi amikor hiba van
	bServiceRun				:BIT;				// 03.8 Szerviz pozícióban a robot, szelep vezérlés mehet.
	
(*-----=== Byte 04 ===-----*)
	_reserved_04			:BYTE;
	
(*-----=== Byte 05 ===-----*)
	bCNC_1_Set				:BIT;				// 05.1	Robot CNC-1-be menne
	bCNC_1_ViseClose_Set	:BIT;				// 05.2	Robot CNC-1 satu zárásra vár
	bCNC_1_ViseOpen_Set		:BIT;				// 05.3	Robot CNC-1 satu nyitásra vár
	bCNC_2_Set				:BIT;				// 05.4	Robot CNC-2-be menne
	bCNC_2_ViseClose_Set	:BIT;				// 05.5	Robot CNC-2 satu zárásra vár
	bCNC_2_ViseOpen_Set		:BIT;				// 05.6	Robot CNC-2 satu nyitásra vár
	bCNC_3_Set				:BIT;				// 05.7	Robot CNC-3-be menne
	bCNC_3_ViseClose_Set	:BIT;				// 05.8	Robot CNC-3 satu zárásra vár
	
(*-----=== Byte 06 ===-----*)
	bCNC_3_ViseOpen_Set		:BIT;				// 06.1	Robot CNC-3 satu nyitásra vár
	bPalette_1_Set			:BIT;				// 06.2	Robot Kiemelő 1-hez menne
	bPalette_2_Set			:BIT;				// 06.3	Robot Kiemelő 2-höz menne
	bPalette_3_Set			:BIT;				// 06.4	Robot Kiemelő 3-hoz menne
	bGripperClosed_Set		:BIT;				// 06.5	Robot megfogó zárás SET
	{attribute 'hide'}
	_reserved_06_06			:BIT;		
	{attribute 'hide'}
	_reserved_06_07			:BIT;	
	{attribute 'hide'}
	_reserved_06_08			:BIT;					
	
(*-----=== Byte 07 ===-----*)
	bNotCorrectPrg			:BIT;				// 07.1	Nem megfelelő mozgási program SET
	bNotProductOnRobot		:BIT;				// 07.2	Mozgási program nem hajtható végre, mert a robotnál nincs termék SET
	bProductOnRobot			:BIT;				// 07.3	Mozgási program nem hajtható végre, mert a robotnál termék van SET
	bGripperOpenError		:BIT;				// 07.4	Megfogó nyitási hiba SET
	bGripperCloseError		:BIT;				// 07.5	Megfogó zárási hiba SET
	bOffsetError			:BIT;				// 07.6 Offset érték hiba SET
	bWeightError			:BIT;				// 07.7 Súly érték hiba  SET
	{attribute 'hide'}
	_reserved_07_08			:BIT;

(*-----=== Byte 08 ===-----*)
	{attribute 'hide'}
	_reserved_08			:BYTE;
	
(*-----=== Byte 09 ===-----*)
	bZone_1_CNC_1			:BIT;				// 09.1	Robot bent a területen. - CNC 1
	bZone_2_CNC_2			:BIT;				// 09.2	Robot bent a területen. - CNC 2
	bZone_3_CNC_3			:BIT;				// 09.3	Robot bent a területen. - CNC 3
	bZone_4_Lifter_1		:BIT;				// 09.4	Robot bent a területen. - Kiemelő 1
	bZone_5_Lifter_2		:BIT;				// 09.5	Robot bent a területen. - Kiemelő 2
	bZone_6_Lifter_3		:BIT;				// 09.6	Robot bent a területen. - Kiemelő 3
	bZone_7_Gudel			:BIT;				// 09.7	Robot bent a területen. - Gudel
	bZone_8_Master			:BIT;				// 09.8	Robot bent a területen. - Master
	
(*-----=== Byte 09 ===-----*)
	bRobotInStrip_1			:BIT;				// 10.1	Robot bent a szalag-1-ben.
	bRobotInStrip_2			:BIT;				// 10.2	Robot bent a szalag-2-ben.
	bRobotInStrip_3			:BIT;				// 10.3	Robot bent a szalag-3-ban.
	{attribute 'hide'}
	_reserved_10_04			:BIT;	
	{attribute 'hide'}
	_reserved_10_05			:BIT;		
	{attribute 'hide'}
	_reserved_10_06			:BIT;	
	{attribute 'hide'}
	_reserved_10_07			:BIT;		
	{attribute 'hide'}
	_reserved_10_08			:BIT;	

(*-----=== Byte 11 - 12 ===-----*)
	{attribute 'hide'}
	_reserved_10_12			:ARRAY[11..12] OF BYTE;				
	
(*-----=== Byte 13 ===-----*)
	nProgramNumber			:BYTE;				// 13. Aktuális program szám Robotban,
	
(*-----=== Byte 14 ===-----*)
	nPointNumber			:BYTE;				// 14. Aktuális pont szám
	
(*-----=== Byte 15 ===-----*)
	bKeyAuto				:BIT;				// 15.1	Robot automata-remote üzemmódban
	bKeyManualT1			:BIT;				// 15.2	Robot kézi üzemmódban - 250 mm/sec max sebesség
	bKeyManualT2			:BIT;				// 15.3	Robot kézi üzemmódban - 100 % sebesség
	bSimInput				:BIT;				// 15.4	Szimulálva (force-olva) Input
	bSimOutput				:BIT;				// 15.5	Szimulálva (force-olva) Output
	{attribute 'hide'}
	_reserved_15_06			:BIT;
	{attribute 'hide'}
	_reserved_15_07			:BIT;		
	{attribute 'hide'}
	_reserved_15_08			:BIT;	
	
(*-----=== Byte 16 ===-----*)
	bControllerEmyStop		:BIT;				// 16.1	Robot kontroller vészgomb
	bTeachPendantEmyStop	:BIT;				// 16.2	Teach Pendant vészgomb
	bDeadman				:BIT;				// 16.3	TP engedélyező gomb
	bFence					:BIT;				// 16.4	Fence
	bRot					:BIT;				// 16.5	Robot olyan területre akar mozogni ahova mechanikusan nem ér el
	bHbk					:BIT;				// 16.6	Robot felütközött, védelem
	bEmyStopExternal		:BIT;				// 16.7	Külső vészgomb (gépi)
	bNoPneumatics			:BIT;				// 16.8	A karon lévő pneumatika nem érzékel levegőt
	
(*-----=== Byte 17 ===-----*)
	bBeltBreak				:BIT;				// 17.1	Robot kontroller vészgomb
	bFalm					:BIT;				// 17.2	Ventilátor hiba
	bServoOff				:BIT;				// 17.3	Kivűlről tiltott SERVO engedélyezés
	bIMSTP					:BIT;				// 17.4	Engedélyező jel vissza adása
	bBEKHLD					:BIT;				// 17.5	
	bUSRALM					:BIT;				// 17.6	
	bSRVDSCNCT				:BIT;				// 17.7	
	bNTED					:BIT;				// 17.8			
	
(*-----=== Byte 18-20 ===-----*)
	{attribute 'hide'}
	_reserved_18_20			:ARRAY [18..20] OF BYTE;	
	
(*-----=== Byte 21-22 ===-----*)
	nOffset_ID				:UINT;				// 21-22. PLC-nek visszaadott offszet érték.
	
(*-----=== Byte 23-24 ===-----*)
	nOffset_X_Whole			:INT;				// 23-24. PLC-nek visszaadott X tengelyű egész szám offszet érték.
	
(*-----=== Byte 25-26 ===-----*)
	nOffset_X_Fractional	:UINT;				// 25-26. PLC-nek visszaadott X tengelyű egész tört offszet érték
	
(*-----=== Byte 27-28 ===-----*)
	nOffset_Y_Whole			:INT;				// 27-28. PLC-nek visszaadott Y tengelyű egész szám offszet érték.
	
(*-----=== Byte 29-30 ===-----*)
	nOffset_Y_Fractional	:UINT;				// 29-30. PLC-nek visszaadott Y tengelyű egész tört offszet érték	
	
(*-----=== Byte 31-32 ===-----*)
	nOffset_Z_Whole			:INT;				// 31-32. PLC-nek visszaadott Z tengelyű egész szám offszet érték.
	
(*-----=== Byte 33-34 ===-----*)
	nOffset_Z_Fractional	:UINT;				// 33-34. PLC-nek visszaadott Z tengelyű egész tört offszet érték	
	
(*-----=== Byte 35-36 ===-----*)
	nOffset_W_Whole			:INT;				// 35-36. PLC-nek visszaadott W tengelyű egész szám offszet érték.
	
(*-----=== Byte 37-38 ===-----*)
	nOffset_W_Fractional	:UINT;				// 37-38. PLC-nek visszaadott W tengelyű egész tört offszet érték
	
(*-----=== Byte 39-40 ===-----*)
	nOffset_P_Whole			:INT;				// 39-40. PLC-nek visszaadott P tengelyű egész szám offszet érték.
	
(*-----=== Byte 41-42 ===-----*)
	nOffset_P_Fractional	:UINT;				// 41-42. PLC-nek visszaadott P tengelyű egész tört offszet érték	
	
(*-----=== Byte 43-44 ===-----*)
	nOffset_R_Whole			:INT;				// 43-44. PLC-nek visszaadott R tengelyű egész szám offszet érték.
	
(*-----=== Byte 45-46 ===-----*)
	nOffset_R_Fractional	:UINT;				// 45-46. PLC-nek visszaadott R tengelyű egész tört offszet érték	
	
(*-----=== Byte 47-64 ===-----*)
	{attribute 'hide'}
	_reserved_47_64			:ARRAY [47..64] OF BYTE;		
END_STRUCT
END_TYPE

// ---- POUs/FBs/FanucCNC/DUTs/U_CNC_Fanuc_Input.TcDUT
TYPE U_CNC_Fanuc_Input :
UNION
	aStdIn		AT %I*		:ARRAY [1..32] OF UINT;
	Status					:ST_CNC_Robot_Status;	
END_UNION
END_TYPE

// ---- POUs/FBs/FanucCNC/DUTs/U_CNC_Fanuc_Output.TcDUT
TYPE U_CNC_Fanuc_Output :
UNION
	aStdOut		AT %Q*		:ARRAY [1..32] OF UINT;
	Control					:ST_CNC_Robot_Control;	
END_UNION
END_TYPE

// ---- POUs/FBs/FanucKardex/DUTs/E_Kardex_Robot_Command.TcDUT
{attribute 'qualified_only'}
{attribute 'strict'}
TYPE E_Kardex_Robot_Command :
(
	NoCommand 				:= 0,
	Home					:= 1,
	Wait					:= 2,
	Service					:= 3,
	Measurement_Kardex 		:= 4,
	Pick_Up_Kardex			:= 5,
	Put_Down_Kardex 		:= 6,
	Pick_Up_Mir 			:= 7,
	Put_Down_Mir			:= 8,
	Pick_Up_Puffer 			:= 9,
	Put_Down_Puffer 		:= 10,
	Pick_Up_Strip			:= 11,
	Put_Down_Strip			:= 12,
	Rotate_In_Strip_3		:= 13
);
END_TYPE

// ---- POUs/FBs/FanucKardex/DUTs/E_Kardex_Robot_Programs.TcTLEO
{attribute 'strict'}
{attribute 'to_string'}
TYPE E_Kardex_Robot_Programs :
(
	NoCommand			:= 0, 	// Amíg "0"-ás a programszám addig nincs mozgási program végrehajtás, vár…
	Home				:= 1,	// Robot Zóna-6-ba megy és bemozog alaphelyzetbe
	Park				:= 2,	// Robot Zóna-6-ba megy és bemozog parkoló pozícióba.
	Service				:= 3,	// Robot elmegy szerviz pozícióba.
	KardexMeasurement	:= 4,	// Robot beméri az aktuális kardex polc koordiátáit.
	KardexPickUp 		:= 11,	// Kardex paletta kiszedés
	KardexPutDown	 	:= 12,	// Kardex paletta lerakás
	Mir_1_PickUp		:= 13,	// MIR-1 paletta kiszedés
	Mir_1_PutDown		:= 14,	// MIR-1 paletta lerakás
	Mir_2_PickUp		:= 15,	// MIR-2 paletta kiszedés
	Mir_2_PutDown		:= 16,	// MIR-2 paletta lerakás
	PufferPickUp 		:= 17,	// Puffer paletta kiszedés
	PufferPutDown		:= 18,	// Puffer paletta lerakás
	Strip_1_PickUp		:= 19,	// Szalag-1 paletta kiszedés
	Strip_1_PutDown		:= 20,	// Szalag-1 paletta lerakás
	Strip_2_PickUp		:= 21,	// Szalag-2 paletta kiszedés
	Strip_2_PutDown		:= 22,	// Szalag-2 paletta lerakás
	Strip_3_PickUp		:= 23,	// Szalag-3 paletta kiszedés
	Strip_3_PutDown		:= 24,	// Szalag-3 paletta lerakás
	Strip_3_Rotate		:= 25	// Szalag-3 paletta forgatás
);
END_TYPE

